   1:  PR[91,1] = PR[90,1] + -4.688;
   1:  PR[91,2] = PR[90,2] + 19.334;
   1:  PR[91,3] = PR[90,3] + 39.259;
   1:L PR[91] R[100]mm/sec CNT100;
   1:  PR[91,1] = PR[90,1] + -5.693;
   1:  PR[91,2] = PR[90,2] + 19.538;
   1:  PR[91,3] = PR[90,3] + 39.268;
   1:L PR[91] R[100]mm/sec CNT100;
   1:  PR[91,1] = PR[90,1] + -6.706;
   1:  PR[91,2] = PR[90,2] + 19.692;
   1:  PR[91,3] = PR[90,3] + 39.276;
   1:L PR[91] R[100]mm/sec CNT100;
   1:  PR[91,1] = PR[90,1] + -7.722;
   1:  PR[91,2] = PR[90,2] + 19.796;
   1:  PR[91,3] = PR[90,3] + 39.284;
   1:L PR[91] R[100]mm/sec CNT100;
   1:  PR[91,1] = PR[90,1] + -8.602;
   1:  PR[91,2] = PR[90,2] + 19.845;
   1:  PR[91,3] = PR[90,3] + 39.293;
   1:L PR[91] R[100]mm/sec CNT100;
   1:  PR[91,1] = PR[90,1] + -9.755;
   1:  PR[91,2] = PR[90,2] + 19.856;
   1:  PR[91,3] = PR[90,3] + 39.300;
   1:L PR[91] R[100]mm/sec CNT100;
   1:  PR[91,1] = PR[90,1] + -10.765;
   1:  PR[91,2] = PR[90,2] + 19.813;
   1:  PR[91,3] = PR[90,3] + 39.309;
   1:L PR[91] R[100]mm/sec CNT100;
   1:  PR[91,1] = PR[90,1] + -11.780;
   1:  PR[91,2] = PR[90,2] + 19.722;
   1:  PR[91,3] = PR[90,3] + 39.317;
   1:L PR[91] R[100]mm/sec CNT100;
   1:  PR[91,1] = PR[90,1] + -12.791;
   1:  PR[91,2] = PR[90,2] + 19.583;
   1:  PR[91,3] = PR[90,3] + 39.326;
   1:L PR[91] R[100]mm/sec CNT100;
   1:  PR[91,1] = PR[90,1] + -13.793;
   1:  PR[91,2] = PR[90,2] + 19.395;
   1:  PR[91,3] = PR[90,3] + 39.334;
   1:L PR[91] R[100]mm/sec CNT100;
   1:  PR[91,1] = PR[90,1] + -14.785;
   1:  PR[91,2] = PR[90,2] + 19.159;
   1:  PR[91,3] = PR[90,3] + 39.342;
   1:L PR[91] R[100]mm/sec CNT100;
   1:  PR[91,1] = PR[90,1] + -15.762;
   1:  PR[91,2] = PR[90,2] + 18.876;
   1:  PR[91,3] = PR[90,3] + 39.351;
   1:L PR[91] R[100]mm/sec CNT100;
   1:  PR[91,1] = PR[90,1] + -16.724;
   1:  PR[91,2] = PR[90,2] + 18.547;
   1:  PR[91,3] = PR[90,3] + 39.359;
   1:L PR[91] R[100]mm/sec CNT100;
   1:  PR[91,1] = PR[90,1] + -17.668;
   1:  PR[91,2] = PR[90,2] + 18.171;
   1:  PR[91,3] = PR[90,3] + 39.367;
   1:L PR[91] R[100]mm/sec CNT100;
   1:  PR[91,1] = PR[90,1] + -18.592;
   1:  PR[91,2] = PR[90,2] + 17.751;
   1:  PR[91,3] = PR[90,3] + 39.376;
   1:L PR[91] R[100]mm/sec CNT100;
   1:  PR[91,1] = PR[90,1] + -19.012;
   1:  PR[91,2] = PR[90,2] + 17.536;
   1:  PR[91,3] = PR[90,3] + 39.384;
   1:L PR[91] R[100]mm/sec CNT100;
   1:  PR[91,1] = PR[90,1] + -19.490;
   1:  PR[91,2] = PR[90,2] + 17.288;
   1:  PR[91,3] = PR[90,3] + 39.388;
   1:L PR[91] R[100]mm/sec CNT100;
   1:  PR[91,1] = PR[90,1] + -20.365;
   1:  PR[91,2] = PR[90,2] + 16.783;
   1:  PR[91,3] = PR[90,3] + 39.392;
   1:L PR[91] R[100]mm/sec CNT100;
   1:  PR[91,1] = PR[90,1] + -21.213;
   1:  PR[91,2] = PR[90,2] + 16.237;
   1:  PR[91,3] = PR[90,3] + 39.400;
   1:L PR[91] R[100]mm/sec CNT100;
   1:  PR[91,1] = PR[90,1] + -22.030;
   1:  PR[91,2] = PR[90,2] + 15.652;
   1:  PR[91,3] = PR[90,3] + 39.409;
   1:L PR[91] R[100]mm/sec CNT100;
   1:  PR[91,1] = PR[90,1] + -22.816;
   1:  PR[91,2] = PR[90,2] + 15.029;
   1:  PR[91,3] = PR[90,3] + 39.417;
   1:L PR[91] R[100]mm/sec CNT100;
   1:  PR[91,1] = PR[90,1] + -23.567;
   1:  PR[91,2] = PR[90,2] + 14.370;
   1:  PR[91,3] = PR[90,3] + 39.425;
   1:L PR[91] R[100]mm/sec CNT100;
   1:  PR[91,1] = PR[90,1] + -24.283;
   1:  PR[91,2] = PR[90,2] + 13.676;
   1:  PR[91,3] = PR[90,3] + 39.433;
   1:L PR[91] R[100]mm/sec CNT100;
   1:  PR[91,1] = PR[90,1] + -24.962;
   1:  PR[91,2] = PR[90,2] + 12.948;
   1:  PR[91,3] = PR[90,3] + 39.441;
   1:L PR[91] R[100]mm/sec CNT100;
   1:  PR[91,1] = PR[90,1] + -25.602;
   1:  PR[91,2] = PR[90,2] + 12.188;
   1:  PR[91,3] = PR[90,3] + 39.449;
   1:L PR[91] R[100]mm/sec CNT100;
   1:  PR[91,1] = PR[90,1] + -26.200;
   1:  PR[91,2] = PR[90,2] + 11.396;
   1:  PR[91,3] = PR[90,3] + 39.457;
   1:L PR[91] R[100]mm/sec CNT100;
   1:  PR[91,1] = PR[90,1] + -26.757;
   1:  PR[91,2] = PR[90,2] + 10.575;
   1:  PR[91,3] = PR[90,3] + 39.466;
   1:L PR[91] R[100]mm/sec CNT100;
   1:  PR[91,1] = PR[90,1] + -27.272;
   1:  PR[91,2] = PR[90,2] + 9.727;
   1:  PR[91,3] = PR[90,3] + 39.474;
   1:L PR[91] R[100]mm/sec CNT100;
   1:  PR[91,1] = PR[90,1] + -27.740;
   1:  PR[91,2] = PR[90,2] + 8.860;
   1:  PR[91,3] = PR[90,3] + 39.482;
   1:L PR[91] R[100]mm/sec CNT100;
   1:  PR[91,1] = PR[90,1] + -28.164;
   1:  PR[91,2] = PR[90,2] + 7.973;
   1:  PR[91,3] = PR[90,3] + 39.490;
   1:L PR[91] R[100]mm/sec CNT100;
   1:  PR[91,1] = PR[90,1] + -28.541;
   1:  PR[91,2] = PR[90,2] + 7.075;
   1:  PR[91,3] = PR[90,3] + 39.498;
   1:L PR[91] R[100]mm/sec CNT100;
   1:  PR[91,1] = PR[90,1] + -28.868;
   1:  PR[91,2] = PR[90,2] + 6.168;
   1:  PR[91,3] = PR[90,3] + 39.506;
   1:L PR[91] R[100]mm/sec CNT100;
   1:  PR[91,1] = PR[90,1] + -29.147;
   1:  PR[91,2] = PR[90,2] + 5.252;
   1:  PR[91,3] = PR[90,3] + 39.514;
   1:L PR[91] R[100]mm/sec CNT100;
   1:  PR[91,1] = PR[90,1] + -29.376;
   1:  PR[91,2] = PR[90,2] + 4.327;
   1:  PR[91,3] = PR[90,3] + 39.521;
   1:L PR[91] R[100]mm/sec CNT100;
   1:  PR[91,1] = PR[90,1] + -29.554;
   1:  PR[91,2] = PR[90,2] + 3.388;
   1:  PR[91,3] = PR[90,3] + 39.529;
   1:L PR[91] R[100]mm/sec CNT100;
   1:  PR[91,1] = PR[90,1] + -29.682;
   1:  PR[91,2] = PR[90,2] + 2.429;
   1:  PR[91,3] = PR[90,3] + 39.537;
   1:L PR[91] R[100]mm/sec CNT100;
   1:  PR[91,1] = PR[90,1] + -29.759;
   1:  PR[91,2] = PR[90,2] + 1.444;
   1:  PR[91,3] = PR[90,3] + 39.545;
   1:L PR[91] R[100]mm/sec CNT100;
   1:  PR[91,1] = PR[90,1] + -29.785;
   1:  PR[91,2] = PR[90,2] + 0.428;
   1:  PR[91,3] = PR[90,3] + 39.553;
   1:L PR[91] R[100]mm/sec CNT100;
   1:  PR[91,1] = PR[90,1] + -29.759;
   1:  PR[91,2] = PR[90,2] + -0.589;
   1:  PR[91,3] = PR[90,3] + 39.561;
   1:L PR[91] R[100]mm/sec CNT100;
   1:  PR[91,1] = PR[90,1] + -29.682;
   1:  PR[91,2] = PR[90,2] + -1.574;
   1:  PR[91,3] = PR[90,3] + 39.569;
   1:L PR[91] R[100]mm/sec CNT100;
   1:  PR[91,1] = PR[90,1] + -29.554;
   1:  PR[91,2] = PR[90,2] + -2.533;
   1:  PR[91,3] = PR[90,3] + 39.578;
   1:L PR[91] R[100]mm/sec CNT100;
   1:  PR[91,1] = PR[90,1] + -29.376;
   1:  PR[91,2] = PR[90,2] + -3.472;
   1:  PR[91,3] = PR[90,3] + 39.585;
   1:L PR[91] R[100]mm/sec CNT100;
   1:  PR[91,1] = PR[90,1] + -29.147;
   1:  PR[91,2] = PR[90,2] + -4.396;
   1:  PR[91,3] = PR[90,3] + 39.593;
   1:L PR[91] R[100]mm/sec CNT100;
   1:  PR[91,1] = PR[90,1] + -28.869;
   1:  PR[91,2] = PR[90,2] + -5.312;
   1:  PR[91,3] = PR[90,3] + 39.601;
   1:L PR[91] R[100]mm/sec CNT100;
   1:  PR[91,1] = PR[90,1] + -28.541;
   1:  PR[91,2] = PR[90,2] + -6.219;
   1:  PR[91,3] = PR[90,3] + 39.609;
   1:L PR[91] R[100]mm/sec CNT100;
   1:  PR[91,1] = PR[90,1] + -28.164;
   1:  PR[91,2] = PR[90,2] + -7.118;
   1:  PR[91,3] = PR[90,3] + 39.617;
   1:L PR[91] R[100]mm/sec CNT100;
   1:  PR[91,1] = PR[90,1] + -27.741;
   1:  PR[91,2] = PR[90,2] + -8.004;
   1:  PR[91,3] = PR[90,3] + 39.625;
   1:L PR[91] R[100]mm/sec CNT100;
   1:  PR[91,1] = PR[90,1] + -27.271;
   1:  PR[91,2] = PR[90,2] + -8.872;
   1:  PR[91,3] = PR[90,3] + 39.633;
   1:L PR[91] R[100]mm/sec CNT100;
   1:  PR[91,1] = PR[90,1] + -26.758;
   1:  PR[91,2] = PR[90,2] + -9.720;
   1:  PR[91,3] = PR[90,3] + 39.641;
   1:L PR[91] R[100]mm/sec CNT100;
   1:  PR[91,1] = PR[90,1] + -26.201;
   1:  PR[91,2] = PR[90,2] + -10.540;
   1:  PR[91,3] = PR[90,3] + 39.649;
   1:L PR[91] R[100]mm/sec CNT100;
   1:  PR[91,1] = PR[90,1] + -25.602;
   1:  PR[91,2] = PR[90,2] + -11.332;
   1:  PR[91,3] = PR[90,3] + 39.657;
   1:L PR[91] R[100]mm/sec CNT100;
   1:  PR[91,1] = PR[90,1] + -24.963;
   1:  PR[91,2] = PR[90,2] + -12.092;
   1:  PR[91,3] = PR[90,3] + 39.665;
   1:L PR[91] R[100]mm/sec CNT100;
   1:  PR[91,1] = PR[90,1] + -24.286;
   1:  PR[91,2] = PR[90,2] + -12.818;
   1:  PR[91,3] = PR[90,3] + 39.673;
   1:L PR[91] R[100]mm/sec CNT100;
   1:  PR[91,1] = PR[90,1] + -23.372;
   1:  PR[91,2] = PR[90,2] + -13.688;
   1:  PR[91,3] = PR[90,3] + 39.681;
   1:L PR[91] R[100]mm/sec CNT100;
   1:  PR[91,1] = PR[90,1] + -22.817;
   1:  PR[91,2] = PR[90,2] + -14.173;
   1:  PR[91,3] = PR[90,3] + 39.691;
   1:L PR[91] R[100]mm/sec CNT100;
   1:  PR[91,1] = PR[90,1] + -22.031;
   1:  PR[91,2] = PR[90,2] + -14.796;
   1:  PR[91,3] = PR[90,3] + 39.697;
   1:L PR[91] R[100]mm/sec CNT100;
   1:  PR[91,1] = PR[90,1] + -21.214;
   1:  PR[91,2] = PR[90,2] + -15.381;
   1:  PR[91,3] = PR[90,3] + 39.706;
   1:L PR[91] R[100]mm/sec CNT100;
   1:  PR[91,1] = PR[90,1] + -20.366;
   1:  PR[91,2] = PR[90,2] + -15.927;
   1:  PR[91,3] = PR[90,3] + 39.714;
   1:L PR[91] R[100]mm/sec CNT100;
   1:  PR[91,1] = PR[90,1] + -19.491;
   1:  PR[91,2] = PR[90,2] + -16.433;
   1:  PR[91,3] = PR[90,3] + 39.722;
   1:L PR[91] R[100]mm/sec CNT100;
   1:  PR[91,1] = PR[90,1] + -19.014;
   1:  PR[91,2] = PR[90,2] + -16.681;
   1:  PR[91,3] = PR[90,3] + 39.730;
   1:L PR[91] R[100]mm/sec CNT100;
   1:  PR[91,1] = PR[90,1] + -18.593;
   1:  PR[91,2] = PR[90,2] + -16.895;
   1:  PR[91,3] = PR[90,3] + 39.735;
   1:L PR[91] R[100]mm/sec CNT100;
   1:  PR[91,1] = PR[90,1] + -17.669;
   1:  PR[91,2] = PR[90,2] + -17.316;
   1:  PR[91,3] = PR[90,3] + 39.738;
   1:L PR[91] R[100]mm/sec CNT100;
   1:  PR[91,1] = PR[90,1] + -16.726;
   1:  PR[91,2] = PR[90,2] + -17.691;
   1:  PR[91,3] = PR[90,3] + 39.747;
   1:L PR[91] R[100]mm/sec CNT100;
   1:  PR[91,1] = PR[90,1] + -15.764;
   1:  PR[91,2] = PR[90,2] + -18.021;
   1:  PR[91,3] = PR[90,3] + 39.755;
   1:L PR[91] R[100]mm/sec CNT100;
   1:  PR[91,1] = PR[90,1] + -14.786;
   1:  PR[91,2] = PR[90,2] + -18.304;
   1:  PR[91,3] = PR[90,3] + 39.763;
   1:L PR[91] R[100]mm/sec CNT100;
   1:  PR[91,1] = PR[90,1] + -13.795;
   1:  PR[91,2] = PR[90,2] + -18.539;
   1:  PR[91,3] = PR[90,3] + 39.772;
   1:L PR[91] R[100]mm/sec CNT100;
   1:  PR[91,1] = PR[90,1] + -12.792;
   1:  PR[91,2] = PR[90,2] + -18.727;
   1:  PR[91,3] = PR[90,3] + 39.780;
   1:L PR[91] R[100]mm/sec CNT100;
   1:  PR[91,1] = PR[90,1] + -11.781;
   1:  PR[91,2] = PR[90,2] + -18.867;
   1:  PR[91,3] = PR[90,3] + 39.788;
   1:L PR[91] R[100]mm/sec CNT100;
   1:  PR[91,1] = PR[90,1] + -10.754;
   1:  PR[91,2] = PR[90,2] + -18.958;
   1:  PR[91,3] = PR[90,3] + 39.797;
   1:L PR[91] R[100]mm/sec CNT100;
   1:  PR[91,1] = PR[90,1] + -9.755;
   1:  PR[91,2] = PR[90,2] + -19.001;
   1:  PR[91,3] = PR[90,3] + 39.805;
   1:L PR[91] R[100]mm/sec CNT100;
   1:  PR[91,1] = PR[90,1] + -8.740;
   1:  PR[91,2] = PR[90,2] + -18.995;
   1:  PR[91,3] = PR[90,3] + 39.813;
   1:L PR[91] R[100]mm/sec CNT100;
   1:  PR[91,1] = PR[90,1] + -7.723;
   1:  PR[91,2] = PR[90,2] + -18.941;
   1:  PR[91,3] = PR[90,3] + 39.821;
   1:L PR[91] R[100]mm/sec CNT100;
   1:  PR[91,1] = PR[90,1] + -6.707;
   1:  PR[91,2] = PR[90,2] + -18.837;
   1:  PR[91,3] = PR[90,3] + 39.830;
   1:L PR[91] R[100]mm/sec CNT100;
   1:  PR[91,1] = PR[90,1] + -5.695;
   1:  PR[91,2] = PR[90,2] + -18.683;
   1:  PR[91,3] = PR[90,3] + 39.838;
   1:L PR[91] R[100]mm/sec CNT100;
   1:  PR[91,1] = PR[90,1] + -4.689;
   1:  PR[91,2] = PR[90,2] + -18.479;
   1:  PR[91,3] = PR[90,3] + 39.846;
   1:L PR[91] R[100]mm/sec CNT100;
   1:  PR[91,1] = PR[90,1] + -3.692;
   1:  PR[91,2] = PR[90,2] + -18.226;
   1:  PR[91,3] = PR[90,3] + 39.855;
   1:L PR[91] R[100]mm/sec CNT100;
   1:  PR[91,1] = PR[90,1] + -2.707;
   1:  PR[91,2] = PR[90,2] + -17.922;
   1:  PR[91,3] = PR[90,3] + 39.863;
   1:L PR[91] R[100]mm/sec CNT100;
   1:  PR[91,1] = PR[90,1] + -1.736;
   1:  PR[91,2] = PR[90,2] + -17.569;
   1:  PR[91,3] = PR[90,3] + 39.872;
   1:L PR[91] R[100]mm/sec CNT100;
   1:  PR[91,1] = PR[90,1] + -1.258;
   1:  PR[91,2] = PR[90,2] + -17.370;
   1:  PR[91,3] = PR[90,3] + 39.880;
   1:L PR[91] R[100]mm/sec CNT100;
   1:  PR[91,1] = PR[90,1] + -0.818;
   1:  PR[91,2] = PR[90,2] + -17.224;
   1:  PR[91,3] = PR[90,3] + 39.884;
   1:L PR[91] R[100]mm/sec CNT100;
   1:  PR[91,1] = PR[90,1] + -0.333;
   1:  PR[91,2] = PR[90,2] + -17.149;
   1:  PR[91,3] = PR[90,3] + 39.888;
   1:L PR[91] R[100]mm/sec CNT100;
   1:  PR[91,1] = PR[90,1] + 0.158;
   1:  PR[91,2] = PR[90,2] + -17.154;
   1:  PR[91,3] = PR[90,3] + 39.892;
   1:L PR[91] R[100]mm/sec CNT100;
   1:  PR[91,1] = PR[90,1] + 0.648;
   1:  PR[91,2] = PR[90,2] + -17.241;
   1:  PR[91,3] = PR[90,3] + 39.896;
   1:L PR[91] R[100]mm/sec CNT100;
   1:  PR[91] = PR[90];
   1:  PR[91,1] = PR[90,1] + 2.126;
   1:  PR[91,2] = PR[90,2] + -18.183;
   1:  PR[91,3] = PR[90,3] + 41.230;
   1:L PR[91] R[100]mm/sec CNT100;
   1:  PR[91,1] = PR[90,1] + 3.017;
   1:  PR[91,2] = PR[90,2] + -18.451;
   1:  PR[91,3] = PR[90,3] + 39.912;
   1:L PR[91] R[100]mm/sec CNT100;
   1:  PR[91,1] = PR[90,1] + 4.031;
   1:  PR[91,2] = PR[90,2] + -18.704;
   1:  PR[91,3] = PR[90,3] + 39.920;
   1:L PR[91] R[100]mm/sec CNT100;
   1:  PR[91,1] = PR[90,1] + 5.334;
   1:  PR[91,2] = PR[90,2] + -18.949;
   1:  PR[91,3] = PR[90,3] + 39.929;
   1:L PR[91] R[100]mm/sec CNT100;
   1:  PR[91,1] = PR[90,1] + 6.089;
   1:  PR[91,2] = PR[90,2] + -19.055;
   1:  PR[91,3] = PR[90,3] + 39.939;
   1:L PR[91] R[100]mm/sec CNT100;
   1:  PR[91,1] = PR[90,1] + 7.125;
   1:  PR[91,2] = PR[90,2] + -19.154;
   1:  PR[91,3] = PR[90,3] + 39.946;
   1:L PR[91] R[100]mm/sec CNT100;
   1:  PR[91,1] = PR[90,1] + 8.161;
   1:  PR[91,2] = PR[90,2] + -19.201;
   1:  PR[91,3] = PR[90,3] + 39.954;
   1:L PR[91] R[100]mm/sec CNT100;
   1:  PR[91,1] = PR[90,1] + 9.195;
   1:  PR[91,2] = PR[90,2] + -19.198;
   1:  PR[91,3] = PR[90,3] + 39.963;
   1:L PR[91] R[100]mm/sec CNT100;
   1:  PR[91,1] = PR[90,1] + 10.227;
   1:  PR[91,2] = PR[90,2] + -19.145;
   1:  PR[91,3] = PR[90,3] + 39.971;
   1:L PR[91] R[100]mm/sec CNT100;
   1:  PR[91,1] = PR[90,1] + 10.777;
   1:  PR[91,2] = PR[90,2] + -19.095;
   1:  PR[91,3] = PR[90,3] + 39.980;
   1:L PR[91] R[100]mm/sec CNT100;
   1:  PR[91,1] = PR[90,1] + 11.243;
   1:  PR[91,2] = PR[90,2] + -19.043;
   1:  PR[91,3] = PR[90,3] + 39.984;
   1:L PR[91] R[100]mm/sec CNT100;
   1:  PR[91,1] = PR[90,1] + 12.258;
   1:  PR[91,2] = PR[90,2] + -18.891;
   1:  PR[91,3] = PR[90,3] + 39.988;
   1:L PR[91] R[100]mm/sec CNT100;
   1:  PR[91,1] = PR[90,1] + 13.258;
   1:  PR[91,2] = PR[90,2] + -18.692;
   1:  PR[91,3] = PR[90,3] + 39.997;
   1:L PR[91] R[100]mm/sec CNT100;
   1:  PR[91,1] = PR[90,1] + 14.244;
   1:  PR[91,2] = PR[90,2] + -18.447;
   1:  PR[91,3] = PR[90,3] + 40.005;
   1:L PR[91] R[100]mm/sec CNT100;
   1:  PR[91,1] = PR[90,1] + 15.213;
   1:  PR[91,2] = PR[90,2] + -18.155;
   1:  PR[91,3] = PR[90,3] + 40.013;
   1:L PR[91] R[100]mm/sec CNT100;
   1:  PR[91,1] = PR[90,1] + 16.164;
   1:  PR[91,2] = PR[90,2] + -17.820;
   1:  PR[91,3] = PR[90,3] + 40.022;
   1:L PR[91] R[100]mm/sec CNT100;
   1:  PR[91,1] = PR[90,1] + 16.987;
   1:  PR[91,2] = PR[90,2] + -17.488;
   1:  PR[91,3] = PR[90,3] + 40.030;
   1:L PR[91] R[100]mm/sec CNT100;
   1:  PR[91,1] = PR[90,1] + 17.948;
   1:  PR[91,2] = PR[90,2] + -17.047;
   1:  PR[91,3] = PR[90,3] + 40.037;
   1:L PR[91] R[100]mm/sec CNT100;
   1:  PR[91,1] = PR[90,1] + 18.881;
   1:  PR[91,2] = PR[90,2] + -16.562;
   1:  PR[91,3] = PR[90,3] + 40.046;
   1:L PR[91] R[100]mm/sec CNT100;
   1:  PR[91,1] = PR[90,1] + 19.757;
   1:  PR[91,2] = PR[90,2] + -16.051;
   1:  PR[91,3] = PR[90,3] + 40.054;
   1:L PR[91] R[100]mm/sec CNT100;
   1:  PR[91,1] = PR[90,1] + 20.606;
   1:  PR[91,2] = PR[90,2] + -15.500;
   1:  PR[91,3] = PR[90,3] + 40.063;
   1:L PR[91] R[100]mm/sec CNT100;
   1:  PR[91,1] = PR[90,1] + 21.424;
   1:  PR[91,2] = PR[90,2] + -14.910;
   1:  PR[91,3] = PR[90,3] + 40.071;
   1:L PR[91] R[100]mm/sec CNT100;
   1:  PR[91,1] = PR[90,1] + 22.211;
   1:  PR[91,2] = PR[90,2] + -14.281;
   1:  PR[91,3] = PR[90,3] + 40.079;
   1:L PR[91] R[100]mm/sec CNT100;
   1:  PR[91,1] = PR[90,1] + 22.964;
   1:  PR[91,2] = PR[90,2] + -13.615;
   1:  PR[91,3] = PR[90,3] + 40.088;
   1:L PR[91] R[100]mm/sec CNT100;
   1:  PR[91,1] = PR[90,1] + 23.681;
   1:  PR[91,2] = PR[90,2] + -12.913;
   1:  PR[91,3] = PR[90,3] + 40.096;
   1:L PR[91] R[100]mm/sec CNT100;
   1:  PR[91,1] = PR[90,1] + 24.360;
   1:  PR[91,2] = PR[90,2] + -12.177;
   1:  PR[91,3] = PR[90,3] + 40.104;
   1:L PR[91] R[100]mm/sec CNT100;
   1:  PR[91,1] = PR[90,1] + 25.001;
   1:  PR[91,2] = PR[90,2] + -11.408;
   1:  PR[91,3] = PR[90,3] + 40.112;
   1:L PR[91] R[100]mm/sec CNT100;
   1:  PR[91,1] = PR[90,1] + 25.600;
   1:  PR[91,2] = PR[90,2] + -10.608;
   1:  PR[91,3] = PR[90,3] + 40.121;
   1:L PR[91] R[100]mm/sec CNT100;
   1:  PR[91,1] = PR[90,1] + 26.158;
   1:  PR[91,2] = PR[90,2] + -9.780;
   1:  PR[91,3] = PR[90,3] + 40.129;
   1:L PR[91] R[100]mm/sec CNT100;
   1:  PR[91,1] = PR[90,1] + 26.393;
   1:  PR[91,2] = PR[90,2] + -9.394;
   1:  PR[91,3] = PR[90,3] + 40.137;
   1:L PR[91] R[100]mm/sec CNT100;
   1:  PR[91,1] = PR[90,1] + 26.672;
   1:  PR[91,2] = PR[90,2] + -8.930;
   1:  PR[91,3] = PR[90,3] + 40.141;
   1:L PR[91] R[100]mm/sec CNT100;
   1:  PR[91,1] = PR[90,1] + 27.142;
   1:  PR[91,2] = PR[90,2] + -8.057;
   1:  PR[91,3] = PR[90,3] + 40.145;
   1:L PR[91] R[100]mm/sec CNT100;
   1:  PR[91,1] = PR[90,1] + 27.565;
   1:  PR[91,2] = PR[90,2] + -7.169;
   1:  PR[91,3] = PR[90,3] + 40.153;
   1:L PR[91] R[100]mm/sec CNT100;
   1:  PR[91,1] = PR[90,1] + 27.941;
   1:  PR[91,2] = PR[90,2] + -6.269;
   1:  PR[91,3] = PR[90,3] + 40.161;
   1:L PR[91] R[100]mm/sec CNT100;
   1:  PR[91,1] = PR[90,1] + 28.268;
   1:  PR[91,2] = PR[90,2] + -5.359;
   1:  PR[91,3] = PR[90,3] + 40.169;
   1:L PR[91] R[100]mm/sec CNT100;
   1:  PR[91,1] = PR[90,1] + 28.546;
   1:  PR[91,2] = PR[90,2] + -4.438;
   1:  PR[91,3] = PR[90,3] + 40.177;
   1:L PR[91] R[100]mm/sec CNT100;
   1:  PR[91,1] = PR[90,1] + 28.774;
   1:  PR[91,2] = PR[90,2] + -3.505;
   1:  PR[91,3] = PR[90,3] + 40.185;
   1:L PR[91] R[100]mm/sec CNT100;
   1:  PR[91,1] = PR[90,1] + 28.952;
   1:  PR[91,2] = PR[90,2] + -2.556;
   1:  PR[91,3] = PR[90,3] + 40.193;
   1:L PR[91] R[100]mm/sec CNT100;
   1:  PR[91,1] = PR[90,1] + 29.080;
   1:  PR[91,2] = PR[90,2] + -1.586;
   1:  PR[91,3] = PR[90,3] + 40.201;
   1:L PR[91] R[100]mm/sec CNT100;
   1:  PR[91,1] = PR[90,1] + 29.157;
   1:  PR[91,2] = PR[90,2] + -0.593;
   1:  PR[91,3] = PR[90,3] + 40.209;
   1:L PR[91] R[100]mm/sec CNT100;
   1:  PR[91,1] = PR[90,1] + 29.181;
   1:  PR[91,2] = PR[90,2] + 0.428;
   1:  PR[91,3] = PR[90,3] + 40.217;
   1:L PR[91] R[100]mm/sec CNT100;
   1:  PR[91,1] = PR[90,1] + 29.157;
   1:  PR[91,2] = PR[90,2] + 1.448;
   1:  PR[91,3] = PR[90,3] + 40.226;
   1:L PR[91] R[100]mm/sec CNT100;
   1:  PR[91,1] = PR[90,1] + 29.080;
   1:  PR[91,2] = PR[90,2] + 2.441;
   1:  PR[91,3] = PR[90,3] + 40.234;
   1:L PR[91] R[100]mm/sec CNT100;
   1:  PR[91,1] = PR[90,1] + 28.952;
   1:  PR[91,2] = PR[90,2] + 3.411;
   1:  PR[91,3] = PR[90,3] + 40.242;
   1:L PR[91] R[100]mm/sec CNT100;
   1:  PR[91,1] = PR[90,1] + 28.774;
   1:  PR[91,2] = PR[90,2] + 4.360;
   1:  PR[91,3] = PR[90,3] + 40.250;
   1:L PR[91] R[100]mm/sec CNT100;
   1:  PR[91,1] = PR[90,1] + 28.546;
   1:  PR[91,2] = PR[90,2] + 5.294;
   1:  PR[91,3] = PR[90,3] + 40.258;
   1:L PR[91] R[100]mm/sec CNT100;
   1:  PR[91,1] = PR[90,1] + 28.268;
   1:  PR[91,2] = PR[90,2] + 6.215;
   1:  PR[91,3] = PR[90,3] + 40.266;
   1:L PR[91] R[100]mm/sec CNT100;
   1:  PR[91,1] = PR[90,1] + 27.941;
   1:  PR[91,2] = PR[90,2] + 7.125;
   1:  PR[91,3] = PR[90,3] + 40.274;
   1:L PR[91] R[100]mm/sec CNT100;
   1:  PR[91,1] = PR[90,1] + 27.771;
   1:  PR[91,2] = PR[90,2] + 7.533;
   1:  PR[91,3] = PR[90,3] + 40.282;
   1:L PR[91] R[100]mm/sec CNT100;
   1:  PR[91,1] = PR[90,1] + 27.565;
   1:  PR[91,2] = PR[90,2] + 8.024;
   1:  PR[91,3] = PR[90,3] + 40.285;
   1:L PR[91] R[100]mm/sec CNT100;
   1:  PR[91,1] = PR[90,1] + 27.141;
   1:  PR[91,2] = PR[90,2] + 8.913;
   1:  PR[91,3] = PR[90,3] + 40.290;
   1:L PR[91] R[100]mm/sec CNT100;
   1:  PR[91,1] = PR[90,1] + 26.672;
   1:  PR[91,2] = PR[90,2] + 9.785;
   1:  PR[91,3] = PR[90,3] + 40.298;
   1:L PR[91] R[100]mm/sec CNT100;
   1:  PR[91,1] = PR[90,1] + 26.158;
   1:  PR[91,2] = PR[90,2] + 10.636;
   1:  PR[91,3] = PR[90,3] + 40.306;
   1:L PR[91] R[100]mm/sec CNT100;
   1:  PR[91,1] = PR[90,1] + 25.600;
   1:  PR[91,2] = PR[90,2] + 11.464;
   1:  PR[91,3] = PR[90,3] + 40.314;
   1:L PR[91] R[100]mm/sec CNT100;
   1:  PR[91,1] = PR[90,1] + 25.230;
   1:  PR[91,2] = PR[90,2] + 11.960;
   1:  PR[91,3] = PR[90,3] + 40.322;
   1:L PR[91] R[100]mm/sec CNT100;
   1:  PR[91,1] = PR[90,1] + 25.001;
   1:  PR[91,2] = PR[90,2] + 12.263;
   1:  PR[91,3] = PR[90,3] + 40.328;
   1:L PR[91] R[100]mm/sec CNT100;
   1:  PR[91,1] = PR[90,1] + 24.360;
   1:  PR[91,2] = PR[90,2] + 13.032;
   1:  PR[91,3] = PR[90,3] + 40.331;
   1:L PR[91] R[100]mm/sec CNT100;
   1:  PR[91,1] = PR[90,1] + 23.680;
   1:  PR[91,2] = PR[90,2] + 13.768;
   1:  PR[91,3] = PR[90,3] + 40.339;
   1:L PR[91] R[100]mm/sec CNT100;
   1:  PR[91,1] = PR[90,1] + 22.963;
   1:  PR[91,2] = PR[90,2] + 14.471;
   1:  PR[91,3] = PR[90,3] + 40.347;
   1:L PR[91] R[100]mm/sec CNT100;
   1:  PR[91,1] = PR[90,1] + 22.210;
   1:  PR[91,2] = PR[90,2] + 15.136;
   1:  PR[91,3] = PR[90,3] + 40.355;
   1:L PR[91] R[100]mm/sec CNT100;
   1:  PR[91,1] = PR[90,1] + 21.549;
   1:  PR[91,2] = PR[90,2] + 15.666;
   1:  PR[91,3] = PR[90,3] + 40.364;
   1:L PR[91] R[100]mm/sec CNT100;
   1:  PR[91,1] = PR[90,1] + 20.603;
   1:  PR[91,2] = PR[90,2] + 16.357;
   1:  PR[91,3] = PR[90,3] + 40.371;
   1:L PR[91] R[100]mm/sec CNT100;
   1:  PR[91,1] = PR[90,1] + 19.756;
   1:  PR[91,2] = PR[90,2] + 16.907;
   1:  PR[91,3] = PR[90,3] + 40.380;
   1:L PR[91] R[100]mm/sec CNT100;
   1:  PR[91,1] = PR[90,1] + 18.879;
   1:  PR[91,2] = PR[90,2] + 17.418;
   1:  PR[91,3] = PR[90,3] + 40.388;
   1:L PR[91] R[100]mm/sec CNT100;
   1:  PR[91,1] = PR[90,1] + 17.947;
   1:  PR[91,2] = PR[90,2] + 17.903;
   1:  PR[91,3] = PR[90,3] + 40.397;
   1:L PR[91] R[100]mm/sec CNT100;
   1:  PR[91,1] = PR[90,1] + 16.986;
   1:  PR[91,2] = PR[90,2] + 18.343;
   1:  PR[91,3] = PR[90,3] + 40.405;
   1:L PR[91] R[100]mm/sec CNT100;
   1:  PR[91,1] = PR[90,1] + 16.163;
   1:  PR[91,2] = PR[90,2] + 18.675;
   1:  PR[91,3] = PR[90,3] + 40.414;
   1:L PR[91] R[100]mm/sec CNT100;
   1:  PR[91,1] = PR[90,1] + 15.212;
   1:  PR[91,2] = PR[90,2] + 19.011;
   1:  PR[91,3] = PR[90,3] + 40.421;
   1:L PR[91] R[100]mm/sec CNT100;
   1:  PR[91,1] = PR[90,1] + 14.243;
   1:  PR[91,2] = PR[90,2] + 19.302;
   1:  PR[91,3] = PR[90,3] + 40.430;
   1:L PR[91] R[100]mm/sec CNT100;
   1:  PR[91,1] = PR[90,1] + 13.257;
   1:  PR[91,2] = PR[90,2] + 19.548;
   1:  PR[91,3] = PR[90,3] + 40.438;
   1:L PR[91] R[100]mm/sec CNT100;
   1:  PR[91,1] = PR[90,1] + 12.254;
   1:  PR[91,2] = PR[90,2] + 19.747;
   1:  PR[91,3] = PR[90,3] + 40.446;
   1:L PR[91] R[100]mm/sec CNT100;
   1:  PR[91,1] = PR[90,1] + 11.852;
   1:  PR[91,2] = PR[90,2] + 19.812;
   1:  PR[91,3] = PR[90,3] + 40.455;
   1:L PR[91] R[100]mm/sec CNT100;
   1:  PR[91,1] = PR[90,1] + 11.247;
   1:  PR[91,2] = PR[90,2] + 19.898;
   1:  PR[91,3] = PR[90,3] + 40.458;
   1:L PR[91] R[100]mm/sec CNT100;
   1:  PR[91,1] = PR[90,1] + 10.223;
   1:  PR[91,2] = PR[90,2] + 20.000;
   1:  PR[91,3] = PR[90,3] + 40.463;
   1:L PR[91] R[100]mm/sec CNT100;
   1:  PR[91,1] = PR[90,1] + 9.192;
   1:  PR[91,2] = PR[90,2] + 20.053;
   1:  PR[91,3] = PR[90,3] + 40.472;
   1:L PR[91] R[100]mm/sec CNT100;
   1:  PR[91,1] = PR[90,1] + 8.600;
   1:  PR[91,2] = PR[90,2] + 20.060;
   1:  PR[91,3] = PR[90,3] + 40.480;
   1:L PR[91] R[100]mm/sec CNT100;
   1:  PR[91,1] = PR[90,1] + 8.163;
   1:  PR[91,2] = PR[90,2] + 20.057;
   1:  PR[91,3] = PR[90,3] + 40.485;
   1:L PR[91] R[100]mm/sec CNT100;
   1:  PR[91,1] = PR[90,1] + 7.124;
   1:  PR[91,2] = PR[90,2] + 20.009;
   1:  PR[91,3] = PR[90,3] + 40.488;
   1:L PR[91] R[100]mm/sec CNT100;
   1:  PR[91,1] = PR[90,1] + 6.089;
   1:  PR[91,2] = PR[90,2] + 19.911;
   1:  PR[91,3] = PR[90,3] + 40.497;
   1:L PR[91] R[100]mm/sec CNT100;
   1:  PR[91,1] = PR[90,1] + 5.058;
   1:  PR[91,2] = PR[90,2] + 19.761;
   1:  PR[91,3] = PR[90,3] + 40.506;
   1:L PR[91] R[100]mm/sec CNT100;
   1:  PR[91,1] = PR[90,1] + 4.033;
   1:  PR[91,2] = PR[90,2] + 19.559;
   1:  PR[91,3] = PR[90,3] + 40.514;
   1:L PR[91] R[100]mm/sec CNT100;
   1:  PR[91,1] = PR[90,1] + 3.017;
   1:  PR[91,2] = PR[90,2] + 19.306;
   1:  PR[91,3] = PR[90,3] + 40.523;
   1:L PR[91] R[100]mm/sec CNT100;
   1:  PR[91,1] = PR[90,1] + 2.013;
   1:  PR[91,2] = PR[90,2] + 19.003;
   1:  PR[91,3] = PR[90,3] + 40.531;
   1:L PR[91] R[100]mm/sec CNT100;
   1:  PR[91,1] = PR[90,1] + 0.710;
   1:  PR[91,2] = PR[90,2] + 18.536;
   1:  PR[91,3] = PR[90,3] + 40.540;
   1:L PR[91] R[100]mm/sec CNT100;
   1:  PR[91,1] = PR[90,1] + 0.230;
   1:  PR[91,2] = PR[90,2] + 18.441;
   1:  PR[91,3] = PR[90,3] + 40.551;
   1:L PR[91] R[100]mm/sec CNT100;
   1:  PR[91,1] = PR[90,1] + -0.255;
   1:  PR[91,2] = PR[90,2] + 18.422;
   1:  PR[91,3] = PR[90,3] + 40.555;
   1:L PR[91] R[100]mm/sec CNT100;
   1:  PR[91,1] = PR[90,1] + -0.742;
   1:  PR[91,2] = PR[90,2] + 18.485;
   1:  PR[91,3] = PR[90,3] + 40.559;
   1:L PR[91] R[100]mm/sec CNT100;
   1:  PR[91,1] = PR[90,1] + -1.178;
   1:  PR[91,2] = PR[90,2] + 18.616;
   1:  PR[91,3] = PR[90,3] + 40.563;
   1:L PR[91] R[100]mm/sec CNT100;
   1:  PR[91,1] = PR[90,1] + -2.363;
   1:  PR[91,2] = PR[90,2] + 19.039;
   1:  PR[91,3] = PR[90,3] + 40.567;
   1:L PR[91] R[100]mm/sec CNT100;
   1:  PR[91,1] = PR[90,1] + -3.255;
   1:  PR[91,2] = PR[90,2] + 19.307;
   1:  PR[91,3] = PR[90,3] + 40.577;
   1:L PR[91] R[100]mm/sec CNT100;
   1:  PR[91,1] = PR[90,1] + -4.269;
   1:  PR[91,2] = PR[90,2] + 19.559;
   1:  PR[91,3] = PR[90,3] + 40.585;
   1:L PR[91] R[100]mm/sec CNT100;
   1:  PR[91,1] = PR[90,1] + -5.571;
   1:  PR[91,2] = PR[90,2] + 19.804;
   1:  PR[91,3] = PR[90,3] + 40.594;
   1:L PR[91] R[100]mm/sec CNT100;
   1:  PR[91,1] = PR[90,1] + -6.327;
   1:  PR[91,2] = PR[90,2] + 19.910;
   1:  PR[91,3] = PR[90,3] + 40.604;
   1:L PR[91] R[100]mm/sec CNT100;
   1:  PR[91,1] = PR[90,1] + -7.363;
   1:  PR[91,2] = PR[90,2] + 20.009;
   1:  PR[91,3] = PR[90,3] + 40.611;
   1:L PR[91] R[100]mm/sec CNT100;
   1:  PR[91,1] = PR[90,1] + -8.399;
   1:  PR[91,2] = PR[90,2] + 20.056;
   1:  PR[91,3] = PR[90,3] + 40.619;
   1:L PR[91] R[100]mm/sec CNT100;
   1:  PR[91,1] = PR[90,1] + -9.433;
   1:  PR[91,2] = PR[90,2] + 20.053;
   1:  PR[91,3] = PR[90,3] + 40.628;
   1:L PR[91] R[100]mm/sec CNT100;
   1:  PR[91,1] = PR[90,1] + -10.465;
   1:  PR[91,2] = PR[90,2] + 20.000;
   1:  PR[91,3] = PR[90,3] + 40.636;
   1:L PR[91] R[100]mm/sec CNT100;
   1:  PR[91,1] = PR[90,1] + -11.016;
   1:  PR[91,2] = PR[90,2] + 19.949;
   1:  PR[91,3] = PR[90,3] + 40.645;
   1:L PR[91] R[100]mm/sec CNT100;
   1:  PR[91,1] = PR[90,1] + -11.481;
   1:  PR[91,2] = PR[90,2] + 19.898;
   1:  PR[91,3] = PR[90,3] + 40.649;
   1:L PR[91] R[100]mm/sec CNT100;
   1:  PR[91,1] = PR[90,1] + -12.496;
   1:  PR[91,2] = PR[90,2] + 19.746;
   1:  PR[91,3] = PR[90,3] + 40.653;
   1:L PR[91] R[100]mm/sec CNT100;
   1:  PR[91,1] = PR[90,1] + -13.497;
   1:  PR[91,2] = PR[90,2] + 19.548;
   1:  PR[91,3] = PR[90,3] + 40.662;
   1:L PR[91] R[100]mm/sec CNT100;
   1:  PR[91,1] = PR[90,1] + -14.482;
   1:  PR[91,2] = PR[90,2] + 19.303;
   1:  PR[91,3] = PR[90,3] + 40.670;
   1:L PR[91] R[100]mm/sec CNT100;
   1:  PR[91,1] = PR[90,1] + -15.453;
   1:  PR[91,2] = PR[90,2] + 19.011;
   1:  PR[91,3] = PR[90,3] + 40.678;
   1:L PR[91] R[100]mm/sec CNT100;
   1:  PR[91,1] = PR[90,1] + -16.239;
   1:  PR[91,2] = PR[90,2] + 18.738;
   1:  PR[91,3] = PR[90,3] + 40.687;
   1:L PR[91] R[100]mm/sec CNT100;
   1:  PR[91,1] = PR[90,1] + -17.226;
   1:  PR[91,2] = PR[90,2] + 18.343;
   1:  PR[91,3] = PR[90,3] + 40.693;
   1:L PR[91] R[100]mm/sec CNT100;
   1:  PR[91,1] = PR[90,1] + -18.186;
   1:  PR[91,2] = PR[90,2] + 17.903;
   1:  PR[91,3] = PR[90,3] + 40.702;
   1:L PR[91] R[100]mm/sec CNT100;
   1:  PR[91,1] = PR[90,1] + -19.119;
   1:  PR[91,2] = PR[90,2] + 17.416;
   1:  PR[91,3] = PR[90,3] + 40.711;
   1:L PR[91] R[100]mm/sec CNT100;
   1:  PR[91,1] = PR[90,1] + -19.995;
   1:  PR[91,2] = PR[90,2] + 16.905;
   1:  PR[91,3] = PR[90,3] + 40.719;
   1:L PR[91] R[100]mm/sec CNT100;
   1:  PR[91,1] = PR[90,1] + -20.844;
   1:  PR[91,2] = PR[90,2] + 16.353;
   1:  PR[91,3] = PR[90,3] + 40.728;
   1:L PR[91] R[100]mm/sec CNT100;
   1:  PR[91,1] = PR[90,1] + -21.663;
   1:  PR[91,2] = PR[90,2] + 15.762;
   1:  PR[91,3] = PR[90,3] + 40.736;
   1:L PR[91] R[100]mm/sec CNT100;
   1:  PR[91,1] = PR[90,1] + -22.450;
   1:  PR[91,2] = PR[90,2] + 15.133;
   1:  PR[91,3] = PR[90,3] + 40.744;
   1:L PR[91] R[100]mm/sec CNT100;
   1:  PR[91,1] = PR[90,1] + -23.203;
   1:  PR[91,2] = PR[90,2] + 14.468;
   1:  PR[91,3] = PR[90,3] + 40.753;
   1:L PR[91] R[100]mm/sec CNT100;
   1:  PR[91,1] = PR[90,1] + -23.920;
   1:  PR[91,2] = PR[90,2] + 13.768;
   1:  PR[91,3] = PR[90,3] + 40.761;
   1:L PR[91] R[100]mm/sec CNT100;
   1:  PR[91,1] = PR[90,1] + -24.599;
   1:  PR[91,2] = PR[90,2] + 13.034;
   1:  PR[91,3] = PR[90,3] + 40.769;
   1:L PR[91] R[100]mm/sec CNT100;
   1:  PR[91,1] = PR[90,1] + -25.240;
   1:  PR[91,2] = PR[90,2] + 12.266;
   1:  PR[91,3] = PR[90,3] + 40.777;
   1:L PR[91] R[100]mm/sec CNT100;
   1:  PR[91,1] = PR[90,1] + -25.469;
   1:  PR[91,2] = PR[90,2] + 11.965;
   1:  PR[91,3] = PR[90,3] + 40.786;
   1:L PR[91] R[100]mm/sec CNT100;
   1:  PR[91,1] = PR[90,1] + -25.839;
   1:  PR[91,2] = PR[90,2] + 11.470;
   1:  PR[91,3] = PR[90,3] + 40.789;
   1:L PR[91] R[100]mm/sec CNT100;
   1:  PR[91,1] = PR[90,1] + -26.397;
   1:  PR[91,2] = PR[90,2] + 10.643;
   1:  PR[91,3] = PR[90,3] + 40.794;
   1:L PR[91] R[100]mm/sec CNT100;
   1:  PR[91,1] = PR[90,1] + -26.911;
   1:  PR[91,2] = PR[90,2] + 9.790;
   1:  PR[91,3] = PR[90,3] + 40.802;
   1:L PR[91] R[100]mm/sec CNT100;
   1:  PR[91,1] = PR[90,1] + -27.380;
   1:  PR[91,2] = PR[90,2] + 8.915;
   1:  PR[91,3] = PR[90,3] + 40.810;
   1:L PR[91] R[100]mm/sec CNT100;
   1:  PR[91,1] = PR[90,1] + -27.803;
   1:  PR[91,2] = PR[90,2] + 8.023;
   1:  PR[91,3] = PR[90,3] + 40.818;
   1:L PR[91] R[100]mm/sec CNT100;
   1:  PR[91,1] = PR[90,1] + -28.179;
   1:  PR[91,2] = PR[90,2] + 7.117;
   1:  PR[91,3] = PR[90,3] + 40.826;
   1:L PR[91] R[100]mm/sec CNT100;
   1:  PR[91,1] = PR[90,1] + -28.507;
   1:  PR[91,2] = PR[90,2] + 6.203;
   1:  PR[91,3] = PR[90,3] + 40.834;
   1:L PR[91] R[100]mm/sec CNT100;
   1:  PR[91,1] = PR[90,1] + -28.785;
   1:  PR[91,2] = PR[90,2] + 5.280;
   1:  PR[91,3] = PR[90,3] + 40.842;
   1:L PR[91] R[100]mm/sec CNT100;
   1:  PR[91,1] = PR[90,1] + -29.013;
   1:  PR[91,2] = PR[90,2] + 4.348;
   1:  PR[91,3] = PR[90,3] + 40.850;
   1:L PR[91] R[100]mm/sec CNT100;
   1:  PR[91,1] = PR[90,1] + -29.191;
   1:  PR[91,2] = PR[90,2] + 3.402;
   1:  PR[91,3] = PR[90,3] + 40.858;
   1:L PR[91] R[100]mm/sec CNT100;
   1:  PR[91,1] = PR[90,1] + -29.319;
   1:  PR[91,2] = PR[90,2] + 2.436;
   1:  PR[91,3] = PR[90,3] + 40.866;
   1:L PR[91] R[100]mm/sec CNT100;
   1:  PR[91,1] = PR[90,1] + -29.396;
   1:  PR[91,2] = PR[90,2] + 1.447;
   1:  PR[91,3] = PR[90,3] + 40.874;
   1:L PR[91] R[100]mm/sec CNT100;
   1:  PR[91,1] = PR[90,1] + -29.420;
   1:  PR[91,2] = PR[90,2] + 0.428;
   1:  PR[91,3] = PR[90,3] + 40.882;
   1:L PR[91] R[100]mm/sec CNT100;
   1:  PR[91,1] = PR[90,1] + -29.396;
   1:  PR[91,2] = PR[90,2] + -0.592;
   1:  PR[91,3] = PR[90,3] + 40.891;
   1:L PR[91] R[100]mm/sec CNT100;
   1:  PR[91,1] = PR[90,1] + -29.319;
   1:  PR[91,2] = PR[90,2] + -1.581;
   1:  PR[91,3] = PR[90,3] + 40.899;
   1:L PR[91] R[100]mm/sec CNT100;
   1:  PR[91,1] = PR[90,1] + -29.191;
   1:  PR[91,2] = PR[90,2] + -2.546;
   1:  PR[91,3] = PR[90,3] + 40.907;
   1:L PR[91] R[100]mm/sec CNT100;
   1:  PR[91,1] = PR[90,1] + -29.013;
   1:  PR[91,2] = PR[90,2] + -3.492;
   1:  PR[91,3] = PR[90,3] + 40.915;
   1:L PR[91] R[100]mm/sec CNT100;
   1:  PR[91,1] = PR[90,1] + -28.785;
   1:  PR[91,2] = PR[90,2] + -4.425;
   1:  PR[91,3] = PR[90,3] + 40.923;
   1:L PR[91] R[100]mm/sec CNT100;
   1:  PR[91,1] = PR[90,1] + -28.507;
   1:  PR[91,2] = PR[90,2] + -5.348;
   1:  PR[91,3] = PR[90,3] + 40.931;
   1:L PR[91] R[100]mm/sec CNT100;
   1:  PR[91,1] = PR[90,1] + -28.179;
   1:  PR[91,2] = PR[90,2] + -6.262;
   1:  PR[91,3] = PR[90,3] + 40.939;
   1:L PR[91] R[100]mm/sec CNT100;
   1:  PR[91,1] = PR[90,1] + -27.803;
   1:  PR[91,2] = PR[90,2] + -7.167;
   1:  PR[91,3] = PR[90,3] + 40.947;
   1:L PR[91] R[100]mm/sec CNT100;
   1:  PR[91,1] = PR[90,1] + -27.380;
   1:  PR[91,2] = PR[90,2] + -8.060;
   1:  PR[91,3] = PR[90,3] + 40.955;
   1:L PR[91] R[100]mm/sec CNT100;
   1:  PR[91,1] = PR[90,1] + -26.910;
   1:  PR[91,2] = PR[90,2] + -8.935;
   1:  PR[91,3] = PR[90,3] + 40.963;
   1:L PR[91] R[100]mm/sec CNT100;
   1:  PR[91,1] = PR[90,1] + -26.633;
   1:  PR[91,2] = PR[90,2] + -9.398;
   1:  PR[91,3] = PR[90,3] + 40.971;
   1:L PR[91] R[100]mm/sec CNT100;
   1:  PR[91,1] = PR[90,1] + -26.397;
   1:  PR[91,2] = PR[90,2] + -9.787;
   1:  PR[91,3] = PR[90,3] + 40.976;
   1:L PR[91] R[100]mm/sec CNT100;
   1:  PR[91,1] = PR[90,1] + -25.840;
   1:  PR[91,2] = PR[90,2] + -10.614;
   1:  PR[91,3] = PR[90,3] + 40.979;
   1:L PR[91] R[100]mm/sec CNT100;
   1:  PR[91,1] = PR[90,1] + -25.240;
   1:  PR[91,2] = PR[90,2] + -11.411;
   1:  PR[91,3] = PR[90,3] + 40.987;
   1:L PR[91] R[100]mm/sec CNT100;
   1:  PR[91,1] = PR[90,1] + -24.600;
   1:  PR[91,2] = PR[90,2] + -12.178;
   1:  PR[91,3] = PR[90,3] + 40.996;
   1:L PR[91] R[100]mm/sec CNT100;
   1:  PR[91,1] = PR[90,1] + -23.920;
   1:  PR[91,2] = PR[90,2] + -12.912;
   1:  PR[91,3] = PR[90,3] + 41.004;
   1:L PR[91] R[100]mm/sec CNT100;
   1:  PR[91,1] = PR[90,1] + -23.203;
   1:  PR[91,2] = PR[90,2] + -13.612;
   1:  PR[91,3] = PR[90,3] + 41.012;
   1:L PR[91] R[100]mm/sec CNT100;
   1:  PR[91,1] = PR[90,1] + -22.451;
   1:  PR[91,2] = PR[90,2] + -14.278;
   1:  PR[91,3] = PR[90,3] + 41.020;
   1:L PR[91] R[100]mm/sec CNT100;
   1:  PR[91,1] = PR[90,1] + -21.664;
   1:  PR[91,2] = PR[90,2] + -14.906;
   1:  PR[91,3] = PR[90,3] + 41.029;
   1:L PR[91] R[100]mm/sec CNT100;
   1:  PR[91,1] = PR[90,1] + -20.845;
   1:  PR[91,2] = PR[90,2] + -15.497;
   1:  PR[91,3] = PR[90,3] + 41.037;
   1:L PR[91] R[100]mm/sec CNT100;
   1:  PR[91,1] = PR[90,1] + -19.996;
   1:  PR[91,2] = PR[90,2] + -16.049;
   1:  PR[91,3] = PR[90,3] + 41.045;
   1:L PR[91] R[100]mm/sec CNT100;
   1:  PR[91,1] = PR[90,1] + -19.119;
   1:  PR[91,2] = PR[90,2] + -16.561;
   1:  PR[91,3] = PR[90,3] + 41.053;
   1:L PR[91] R[100]mm/sec CNT100;
   1:  PR[91,1] = PR[90,1] + -18.187;
   1:  PR[91,2] = PR[90,2] + -17.047;
   1:  PR[91,3] = PR[90,3] + 41.062;
   1:L PR[91] R[100]mm/sec CNT100;
   1:  PR[91,1] = PR[90,1] + -17.226;
   1:  PR[91,2] = PR[90,2] + -17.488;
   1:  PR[91,3] = PR[90,3] + 41.070;
   1:L PR[91] R[100]mm/sec CNT100;
   1:  PR[91,1] = PR[90,1] + -16.403;
   1:  PR[91,2] = PR[90,2] + -17.821;
   1:  PR[91,3] = PR[90,3] + 41.079;
   1:L PR[91] R[100]mm/sec CNT100;
   1:  PR[91,1] = PR[90,1] + -15.452;
   1:  PR[91,2] = PR[90,2] + -18.156;
   1:  PR[91,3] = PR[90,3] + 41.086;
   1:L PR[91] R[100]mm/sec CNT100;
   1:  PR[91,1] = PR[90,1] + -14.483;
   1:  PR[91,2] = PR[90,2] + -18.447;
   1:  PR[91,3] = PR[90,3] + 41.095;
   1:L PR[91] R[100]mm/sec CNT100;
   1:  PR[91,1] = PR[90,1] + -13.498;
   1:  PR[91,2] = PR[90,2] + -18.692;
   1:  PR[91,3] = PR[90,3] + 41.103;
   1:L PR[91] R[100]mm/sec CNT100;
   1:  PR[91,1] = PR[90,1] + -12.494;
   1:  PR[91,2] = PR[90,2] + -18.892;
   1:  PR[91,3] = PR[90,3] + 41.111;
   1:L PR[91] R[100]mm/sec CNT100;
   1:  PR[91,1] = PR[90,1] + -12.093;
   1:  PR[91,2] = PR[90,2] + -18.957;
   1:  PR[91,3] = PR[90,3] + 41.120;
   1:L PR[91] R[100]mm/sec CNT100;
   1:  PR[91,1] = PR[90,1] + -11.488;
   1:  PR[91,2] = PR[90,2] + -19.042;
   1:  PR[91,3] = PR[90,3] + 41.123;
   1:L PR[91] R[100]mm/sec CNT100;
   1:  PR[91,1] = PR[90,1] + -10.463;
   1:  PR[91,2] = PR[90,2] + -19.145;
   1:  PR[91,3] = PR[90,3] + 41.128;
   1:L PR[91] R[100]mm/sec CNT100;
   1:  PR[91,1] = PR[90,1] + -9.432;
   1:  PR[91,2] = PR[90,2] + -19.198;
   1:  PR[91,3] = PR[90,3] + 41.137;
   1:L PR[91] R[100]mm/sec CNT100;
   1:  PR[91,1] = PR[90,1] + -8.840;
   1:  PR[91,2] = PR[90,2] + -19.204;
   1:  PR[91,3] = PR[90,3] + 41.145;
   1:L PR[91] R[100]mm/sec CNT100;
   1:  PR[91,1] = PR[90,1] + -8.403;
   1:  PR[91,2] = PR[90,2] + -19.201;
   1:  PR[91,3] = PR[90,3] + 41.150;
   1:L PR[91] R[100]mm/sec CNT100;
   1:  PR[91,1] = PR[90,1] + -7.364;
   1:  PR[91,2] = PR[90,2] + -19.154;
   1:  PR[91,3] = PR[90,3] + 41.153;
   1:L PR[91] R[100]mm/sec CNT100;
   1:  PR[91,1] = PR[90,1] + -6.328;
   1:  PR[91,2] = PR[90,2] + -19.055;
   1:  PR[91,3] = PR[90,3] + 41.162;
   1:L PR[91] R[100]mm/sec CNT100;
   1:  PR[91,1] = PR[90,1] + -5.573;
   1:  PR[91,2] = PR[90,2] + -18.949;
   1:  PR[91,3] = PR[90,3] + 41.171;
   1:L PR[91] R[100]mm/sec CNT100;
   1:  PR[91,1] = PR[90,1] + -4.269;
   1:  PR[91,2] = PR[90,2] + -18.704;
   1:  PR[91,3] = PR[90,3] + 41.177;
   1:L PR[91] R[100]mm/sec CNT100;
   1:  PR[91,1] = PR[90,1] + -3.255;
   1:  PR[91,2] = PR[90,2] + -18.453;
   1:  PR[91,3] = PR[90,3] + 41.188;
   1:L PR[91] R[100]mm/sec CNT100;
   1:  PR[91,1] = PR[90,1] + -2.364;
   1:  PR[91,2] = PR[90,2] + -18.184;
   1:  PR[91,3] = PR[90,3] + 41.196;
   1:L PR[91] R[100]mm/sec CNT100;
   1:  PR[91,1] = PR[90,1] + -1.178;
   1:  PR[91,2] = PR[90,2] + -17.761;
   1:  PR[91,3] = PR[90,3] + 41.204;
   1:L PR[91] R[100]mm/sec CNT100;
   1:  PR[91,1] = PR[90,1] + -0.741;
   1:  PR[91,2] = PR[90,2] + -17.630;
   1:  PR[91,3] = PR[90,3] + 41.214;
   1:L PR[91] R[100]mm/sec CNT100;
   1:  PR[91,1] = PR[90,1] + -0.255;
   1:  PR[91,2] = PR[90,2] + -17.567;
   1:  PR[91,3] = PR[90,3] + 41.218;
   1:L PR[91] R[100]mm/sec CNT100;
   1:  PR[91,1] = PR[90,1] + 0.235;
   1:  PR[91,2] = PR[90,2] + -17.586;
   1:  PR[91,3] = PR[90,3] + 41.222;
   1:L PR[91] R[100]mm/sec CNT100;
   1:  PR[91,1] = PR[90,1] + 0.709;
   1:  PR[91,2] = PR[90,2] + -17.680;
   1:  PR[91,3] = PR[90,3] + 41.226;
   1:L PR[91] R[100]mm/sec CNT100;
   1:  PR[91] = PR[90];
   1:  PR[91,1] = PR[90,1] + 1.518;
   1:  PR[91,2] = PR[90,2] + -18.372;
   1:  PR[91,3] = PR[90,3] + 42.560;
   1:L PR[91] R[100]mm/sec CNT100;
   1:  PR[91,1] = PR[90,1] + 2.539;
   1:  PR[91,2] = PR[90,2] + -18.676;
   1:  PR[91,3] = PR[90,3] + 41.237;
   1:L PR[91] R[100]mm/sec CNT100;
   1:  PR[91,1] = PR[90,1] + 3.575;
   1:  PR[91,2] = PR[90,2] + -18.929;
   1:  PR[91,3] = PR[90,3] + 41.245;
   1:L PR[91] R[100]mm/sec CNT100;
   1:  PR[91,1] = PR[90,1] + 4.622;
   1:  PR[91,2] = PR[90,2] + -19.129;
   1:  PR[91,3] = PR[90,3] + 41.254;
   1:L PR[91] R[100]mm/sec CNT100;
   1:  PR[91,1] = PR[90,1] + 5.679;
   1:  PR[91,2] = PR[90,2] + -19.276;
   1:  PR[91,3] = PR[90,3] + 41.263;
   1:L PR[91] R[100]mm/sec CNT100;
   1:  PR[91,1] = PR[90,1] + 6.741;
   1:  PR[91,2] = PR[90,2] + -19.369;
   1:  PR[91,3] = PR[90,3] + 41.272;
   1:L PR[91] R[100]mm/sec CNT100;
   1:  PR[91,1] = PR[90,1] + 7.807;
   1:  PR[91,2] = PR[90,2] + -19.409;
   1:  PR[91,3] = PR[90,3] + 41.281;
   1:L PR[91] R[100]mm/sec CNT100;
   1:  PR[91,1] = PR[90,1] + 8.873;
   1:  PR[91,2] = PR[90,2] + -19.396;
   1:  PR[91,3] = PR[90,3] + 41.289;
   1:L PR[91] R[100]mm/sec CNT100;
   1:  PR[91,1] = PR[90,1] + 9.921;
   1:  PR[91,2] = PR[90,2] + -19.332;
   1:  PR[91,3] = PR[90,3] + 41.298;
   1:L PR[91] R[100]mm/sec CNT100;
   1:  PR[91,1] = PR[90,1] + 11.069;
   1:  PR[91,2] = PR[90,2] + -19.203;
   1:  PR[91,3] = PR[90,3] + 41.307;
   1:L PR[91] R[100]mm/sec CNT100;
   1:  PR[91,1] = PR[90,1] + 11.991;
   1:  PR[91,2] = PR[90,2] + -19.054;
   1:  PR[91,3] = PR[90,3] + 41.316;
   1:L PR[91] R[100]mm/sec CNT100;
   1:  PR[91,1] = PR[90,1] + 13.008;
   1:  PR[91,2] = PR[90,2] + -18.840;
   1:  PR[91,3] = PR[90,3] + 41.324;
   1:L PR[91] R[100]mm/sec CNT100;
   1:  PR[91,1] = PR[90,1] + 14.009;
   1:  PR[91,2] = PR[90,2] + -18.578;
   1:  PR[91,3] = PR[90,3] + 41.333;
   1:L PR[91] R[100]mm/sec CNT100;
   1:  PR[91,1] = PR[90,1] + 14.993;
   1:  PR[91,2] = PR[90,2] + -18.269;
   1:  PR[91,3] = PR[90,3] + 41.341;
   1:L PR[91] R[100]mm/sec CNT100;
   1:  PR[91,1] = PR[90,1] + 15.958;
   1:  PR[91,2] = PR[90,2] + -17.915;
   1:  PR[91,3] = PR[90,3] + 41.350;
   1:L PR[91] R[100]mm/sec CNT100;
   1:  PR[91,1] = PR[90,1] + 16.900;
   1:  PR[91,2] = PR[90,2] + -17.516;
   1:  PR[91,3] = PR[90,3] + 41.358;
   1:L PR[91] R[100]mm/sec CNT100;
   1:  PR[91,1] = PR[90,1] + 17.818;
   1:  PR[91,2] = PR[90,2] + -17.075;
   1:  PR[91,3] = PR[90,3] + 41.367;
   1:L PR[91] R[100]mm/sec CNT100;
   1:  PR[91,1] = PR[90,1] + 18.710;
   1:  PR[91,2] = PR[90,2] + -16.593;
   1:  PR[91,3] = PR[90,3] + 41.375;
   1:L PR[91] R[100]mm/sec CNT100;
   1:  PR[91,1] = PR[90,1] + 19.574;
   1:  PR[91,2] = PR[90,2] + -16.070;
   1:  PR[91,3] = PR[90,3] + 41.384;
   1:L PR[91] R[100]mm/sec CNT100;
   1:  PR[91,1] = PR[90,1] + 20.411;
   1:  PR[91,2] = PR[90,2] + -15.507;
   1:  PR[91,3] = PR[90,3] + 41.392;
   1:L PR[91] R[100]mm/sec CNT100;
   1:  PR[91,1] = PR[90,1] + 20.913;
   1:  PR[91,2] = PR[90,2] + -15.144;
   1:  PR[91,3] = PR[90,3] + 41.400;
   1:L PR[91] R[100]mm/sec CNT100;
   1:  PR[91,1] = PR[90,1] + 21.733;
   1:  PR[91,2] = PR[90,2] + -14.492;
   1:  PR[91,3] = PR[90,3] + 41.405;
   1:L PR[91] R[100]mm/sec CNT100;
   1:  PR[91,1] = PR[90,1] + 22.513;
   1:  PR[91,2] = PR[90,2] + -13.804;
   1:  PR[91,3] = PR[90,3] + 41.414;
   1:L PR[91] R[100]mm/sec CNT100;
   1:  PR[91,1] = PR[90,1] + 23.254;
   1:  PR[91,2] = PR[90,2] + -13.080;
   1:  PR[91,3] = PR[90,3] + 41.423;
   1:L PR[91] R[100]mm/sec CNT100;
   1:  PR[91,1] = PR[90,1] + 23.952;
   1:  PR[91,2] = PR[90,2] + -12.323;
   1:  PR[91,3] = PR[90,3] + 41.431;
   1:L PR[91] R[100]mm/sec CNT100;
   1:  PR[91,1] = PR[90,1] + 24.608;
   1:  PR[91,2] = PR[90,2] + -11.534;
   1:  PR[91,3] = PR[90,3] + 41.440;
   1:L PR[91] R[100]mm/sec CNT100;
   1:  PR[91,1] = PR[90,1] + 25.219;
   1:  PR[91,2] = PR[90,2] + -10.716;
   1:  PR[91,3] = PR[90,3] + 41.448;
   1:L PR[91] R[100]mm/sec CNT100;
   1:  PR[91,1] = PR[90,1] + 25.786;
   1:  PR[91,2] = PR[90,2] + -9.871;
   1:  PR[91,3] = PR[90,3] + 41.457;
   1:L PR[91] R[100]mm/sec CNT100;
   1:  PR[91,1] = PR[90,1] + 26.306;
   1:  PR[91,2] = PR[90,2] + -9.005;
   1:  PR[91,3] = PR[90,3] + 41.465;
   1:L PR[91] R[100]mm/sec CNT100;
   1:  PR[91,1] = PR[90,1] + 26.789;
   1:  PR[91,2] = PR[90,2] + -8.100;
   1:  PR[91,3] = PR[90,3] + 41.473;
   1:L PR[91] R[100]mm/sec CNT100;
   1:  PR[91,1] = PR[90,1] + 27.208;
   1:  PR[91,2] = PR[90,2] + -7.213;
   1:  PR[91,3] = PR[90,3] + 41.482;
   1:L PR[91] R[100]mm/sec CNT100;
   1:  PR[91,1] = PR[90,1] + 27.582;
   1:  PR[91,2] = PR[90,2] + -6.313;
   1:  PR[91,3] = PR[90,3] + 41.490;
   1:L PR[91] R[100]mm/sec CNT100;
   1:  PR[91,1] = PR[90,1] + 27.909;
   1:  PR[91,2] = PR[90,2] + -5.396;
   1:  PR[91,3] = PR[90,3] + 41.498;
   1:L PR[91] R[100]mm/sec CNT100;
   1:  PR[91,1] = PR[90,1] + 28.187;
   1:  PR[91,2] = PR[90,2] + -4.467;
   1:  PR[91,3] = PR[90,3] + 41.506;
   1:L PR[91] R[100]mm/sec CNT100;
   1:  PR[91,1] = PR[90,1] + 28.416;
   1:  PR[91,2] = PR[90,2] + -3.526;
   1:  PR[91,3] = PR[90,3] + 41.514;
   1:L PR[91] R[100]mm/sec CNT100;
   1:  PR[91,1] = PR[90,1] + 28.594;
   1:  PR[91,2] = PR[90,2] + -2.569;
   1:  PR[91,3] = PR[90,3] + 41.522;
   1:L PR[91] R[100]mm/sec CNT100;
   1:  PR[91,1] = PR[90,1] + 28.722;
   1:  PR[91,2] = PR[90,2] + -1.594;
   1:  PR[91,3] = PR[90,3] + 41.530;
   1:L PR[91] R[100]mm/sec CNT100;
   1:  PR[91,1] = PR[90,1] + 28.799;
   1:  PR[91,2] = PR[90,2] + -0.596;
   1:  PR[91,3] = PR[90,3] + 41.538;
   1:L PR[91] R[100]mm/sec CNT100;
   1:  PR[91,1] = PR[90,1] + 28.824;
   1:  PR[91,2] = PR[90,2] + 0.428;
   1:  PR[91,3] = PR[90,3] + 41.547;
   1:L PR[91] R[100]mm/sec CNT100;
   1:  PR[91,1] = PR[90,1] + 28.799;
   1:  PR[91,2] = PR[90,2] + 1.451;
   1:  PR[91,3] = PR[90,3] + 41.555;
   1:L PR[91] R[100]mm/sec CNT100;
   1:  PR[91,1] = PR[90,1] + 28.722;
   1:  PR[91,2] = PR[90,2] + 2.449;
   1:  PR[91,3] = PR[90,3] + 41.563;
   1:L PR[91] R[100]mm/sec CNT100;
   1:  PR[91,1] = PR[90,1] + 28.594;
   1:  PR[91,2] = PR[90,2] + 3.425;
   1:  PR[91,3] = PR[90,3] + 41.572;
   1:L PR[91] R[100]mm/sec CNT100;
   1:  PR[91,1] = PR[90,1] + 28.416;
   1:  PR[91,2] = PR[90,2] + 4.382;
   1:  PR[91,3] = PR[90,3] + 41.580;
   1:L PR[91] R[100]mm/sec CNT100;
   1:  PR[91,1] = PR[90,1] + 28.187;
   1:  PR[91,2] = PR[90,2] + 5.323;
   1:  PR[91,3] = PR[90,3] + 41.588;
   1:L PR[91] R[100]mm/sec CNT100;
   1:  PR[91,1] = PR[90,1] + 27.909;
   1:  PR[91,2] = PR[90,2] + 6.251;
   1:  PR[91,3] = PR[90,3] + 41.596;
   1:L PR[91] R[100]mm/sec CNT100;
   1:  PR[91,1] = PR[90,1] + 27.582;
   1:  PR[91,2] = PR[90,2] + 7.168;
   1:  PR[91,3] = PR[90,3] + 41.604;
   1:L PR[91] R[100]mm/sec CNT100;
   1:  PR[91,1] = PR[90,1] + 27.205;
   1:  PR[91,2] = PR[90,2] + 8.075;
   1:  PR[91,3] = PR[90,3] + 41.612;
   1:L PR[91] R[100]mm/sec CNT100;
   1:  PR[91,1] = PR[90,1] + 26.780;
   1:  PR[91,2] = PR[90,2] + 8.974;
   1:  PR[91,3] = PR[90,3] + 41.620;
   1:L PR[91] R[100]mm/sec CNT100;
   1:  PR[91,1] = PR[90,1] + 26.306;
   1:  PR[91,2] = PR[90,2] + 9.860;
   1:  PR[91,3] = PR[90,3] + 41.628;
   1:L PR[91] R[100]mm/sec CNT100;
   1:  PR[91,1] = PR[90,1] + 25.785;
   1:  PR[91,2] = PR[90,2] + 10.728;
   1:  PR[91,3] = PR[90,3] + 41.637;
   1:L PR[91] R[100]mm/sec CNT100;
   1:  PR[91,1] = PR[90,1] + 25.286;
   1:  PR[91,2] = PR[90,2] + 11.473;
   1:  PR[91,3] = PR[90,3] + 41.645;
   1:L PR[91] R[100]mm/sec CNT100;
   1:  PR[91,1] = PR[90,1] + 24.607;
   1:  PR[91,2] = PR[90,2] + 12.391;
   1:  PR[91,3] = PR[90,3] + 41.652;
   1:L PR[91] R[100]mm/sec CNT100;
   1:  PR[91,1] = PR[90,1] + 23.952;
   1:  PR[91,2] = PR[90,2] + 13.179;
   1:  PR[91,3] = PR[90,3] + 41.662;
   1:L PR[91] R[100]mm/sec CNT100;
   1:  PR[91,1] = PR[90,1] + 23.253;
   1:  PR[91,2] = PR[90,2] + 13.936;
   1:  PR[91,3] = PR[90,3] + 41.670;
   1:L PR[91] R[100]mm/sec CNT100;
   1:  PR[91,1] = PR[90,1] + 22.513;
   1:  PR[91,2] = PR[90,2] + 14.660;
   1:  PR[91,3] = PR[90,3] + 41.679;
   1:L PR[91] R[100]mm/sec CNT100;
   1:  PR[91,1] = PR[90,1] + 21.733;
   1:  PR[91,2] = PR[90,2] + 15.347;
   1:  PR[91,3] = PR[90,3] + 41.687;
   1:L PR[91] R[100]mm/sec CNT100;
   1:  PR[91,1] = PR[90,1] + 20.912;
   1:  PR[91,2] = PR[90,2] + 15.999;
   1:  PR[91,3] = PR[90,3] + 41.696;
   1:L PR[91] R[100]mm/sec CNT100;
   1:  PR[91,1] = PR[90,1] + 20.407;
   1:  PR[91,2] = PR[90,2] + 16.366;
   1:  PR[91,3] = PR[90,3] + 41.705;
   1:L PR[91] R[100]mm/sec CNT100;
   1:  PR[91,1] = PR[90,1] + 20.061;
   1:  PR[91,2] = PR[90,2] + 16.608;
   1:  PR[91,3] = PR[90,3] + 41.710;
   1:L PR[91] R[100]mm/sec CNT100;
   1:  PR[91,1] = PR[90,1] + 19.168;
   1:  PR[91,2] = PR[90,2] + 17.180;
   1:  PR[91,3] = PR[90,3] + 41.713;
   1:L PR[91] R[100]mm/sec CNT100;
   1:  PR[91,1] = PR[90,1] + 18.244;
   1:  PR[91,2] = PR[90,2] + 17.708;
   1:  PR[91,3] = PR[90,3] + 41.722;
   1:L PR[91] R[100]mm/sec CNT100;
   1:  PR[91,1] = PR[90,1] + 17.291;
   1:  PR[91,2] = PR[90,2] + 18.191;
   1:  PR[91,3] = PR[90,3] + 41.731;
   1:L PR[91] R[100]mm/sec CNT100;
   1:  PR[91,1] = PR[90,1] + 16.304;
   1:  PR[91,2] = PR[90,2] + 18.630;
   1:  PR[91,3] = PR[90,3] + 41.740;
   1:L PR[91] R[100]mm/sec CNT100;
   1:  PR[91,1] = PR[90,1] + 15.962;
   1:  PR[91,2] = PR[90,2] + 18.769;
   1:  PR[91,3] = PR[90,3] + 41.749;
   1:L PR[91] R[100]mm/sec CNT100;
   1:  PR[91,1] = PR[90,1] + 14.993;
   1:  PR[91,2] = PR[90,2] + 19.125;
   1:  PR[91,3] = PR[90,3] + 41.752;
   1:L PR[91] R[100]mm/sec CNT100;
   1:  PR[91,1] = PR[90,1] + 14.009;
   1:  PR[91,2] = PR[90,2] + 19.433;
   1:  PR[91,3] = PR[90,3] + 41.760;
   1:L PR[91] R[100]mm/sec CNT100;
   1:  PR[91,1] = PR[90,1] + 13.007;
   1:  PR[91,2] = PR[90,2] + 19.695;
   1:  PR[91,3] = PR[90,3] + 41.769;
   1:L PR[91] R[100]mm/sec CNT100;
   1:  PR[91,1] = PR[90,1] + 12.152;
   1:  PR[91,2] = PR[90,2] + 19.878;
   1:  PR[91,3] = PR[90,3] + 41.777;
   1:L PR[91] R[100]mm/sec CNT100;
   1:  PR[91,1] = PR[90,1] + 10.960;
   1:  PR[91,2] = PR[90,2] + 20.073;
   1:  PR[91,3] = PR[90,3] + 41.785;
   1:L PR[91] R[100]mm/sec CNT100;
   1:  PR[91,1] = PR[90,1] + 9.922;
   1:  PR[91,2] = PR[90,2] + 20.187;
   1:  PR[91,3] = PR[90,3] + 41.794;
   1:L PR[91] R[100]mm/sec CNT100;
   1:  PR[91,1] = PR[90,1] + 8.869;
   1:  PR[91,2] = PR[90,2] + 20.251;
   1:  PR[91,3] = PR[90,3] + 41.803;
   1:L PR[91] R[100]mm/sec CNT100;
   1:  PR[91,1] = PR[90,1] + 7.806;
   1:  PR[91,2] = PR[90,2] + 20.264;
   1:  PR[91,3] = PR[90,3] + 41.812;
   1:L PR[91] R[100]mm/sec CNT100;
   1:  PR[91,1] = PR[90,1] + 6.741;
   1:  PR[91,2] = PR[90,2] + 20.224;
   1:  PR[91,3] = PR[90,3] + 41.821;
   1:L PR[91] R[100]mm/sec CNT100;
   1:  PR[91,1] = PR[90,1] + 5.679;
   1:  PR[91,2] = PR[90,2] + 20.131;
   1:  PR[91,3] = PR[90,3] + 41.829;
   1:L PR[91] R[100]mm/sec CNT100;
   1:  PR[91,1] = PR[90,1] + 4.622;
   1:  PR[91,2] = PR[90,2] + 19.984;
   1:  PR[91,3] = PR[90,3] + 41.838;
   1:L PR[91] R[100]mm/sec CNT100;
   1:  PR[91,1] = PR[90,1] + 3.575;
   1:  PR[91,2] = PR[90,2] + 19.784;
   1:  PR[91,3] = PR[90,3] + 41.847;
   1:L PR[91] R[100]mm/sec CNT100;
   1:  PR[91,1] = PR[90,1] + 2.539;
   1:  PR[91,2] = PR[90,2] + 19.532;
   1:  PR[91,3] = PR[90,3] + 41.856;
   1:L PR[91] R[100]mm/sec CNT100;
   1:  PR[91,1] = PR[90,1] + 1.517;
   1:  PR[91,2] = PR[90,2] + 19.227;
   1:  PR[91,3] = PR[90,3] + 41.865;
   1:L PR[91] R[100]mm/sec CNT100;
   1:  PR[91,1] = PR[90,1] + 0.774;
   1:  PR[91,2] = PR[90,2] + 18.968;
   1:  PR[91,3] = PR[90,3] + 41.874;
   1:L PR[91] R[100]mm/sec CNT100;
   1:  PR[91,1] = PR[90,1] + 0.310;
   1:  PR[91,2] = PR[90,2] + 18.861;
   1:  PR[91,3] = PR[90,3] + 41.880;
   1:L PR[91] R[100]mm/sec CNT100;
   1:  PR[91,1] = PR[90,1] + -0.180;
   1:  PR[91,2] = PR[90,2] + 18.832;
   1:  PR[91,3] = PR[90,3] + 41.884;
   1:L PR[91] R[100]mm/sec CNT100;
   1:  PR[91,1] = PR[90,1] + -0.666;
   1:  PR[91,2] = PR[90,2] + 18.881;
   1:  PR[91,3] = PR[90,3] + 41.888;
   1:L PR[91] R[100]mm/sec CNT100;
   1:  PR[91,1] = PR[90,1] + -1.112;
   1:  PR[91,2] = PR[90,2] + 19.002;
   1:  PR[91,3] = PR[90,3] + 41.892;
   1:L PR[91] R[100]mm/sec CNT100;
   1:  PR[91,1] = PR[90,1] + -1.754;
   1:  PR[91,2] = PR[90,2] + 19.228;
   1:  PR[91,3] = PR[90,3] + 41.896;
   1:L PR[91] R[100]mm/sec CNT100;
   1:  PR[91,1] = PR[90,1] + -2.776;
   1:  PR[91,2] = PR[90,2] + 19.532;
   1:  PR[91,3] = PR[90,3] + 41.901;
   1:L PR[91] R[100]mm/sec CNT100;
   1:  PR[91,1] = PR[90,1] + -3.812;
   1:  PR[91,2] = PR[90,2] + 19.784;
   1:  PR[91,3] = PR[90,3] + 41.910;
   1:L PR[91] R[100]mm/sec CNT100;
   1:  PR[91,1] = PR[90,1] + -4.860;
   1:  PR[91,2] = PR[90,2] + 19.984;
   1:  PR[91,3] = PR[90,3] + 41.919;
   1:L PR[91] R[100]mm/sec CNT100;
   1:  PR[91,1] = PR[90,1] + -5.916;
   1:  PR[91,2] = PR[90,2] + 20.130;
   1:  PR[91,3] = PR[90,3] + 41.928;
   1:L PR[91] R[100]mm/sec CNT100;
   1:  PR[91,1] = PR[90,1] + -6.979;
   1:  PR[91,2] = PR[90,2] + 20.224;
   1:  PR[91,3] = PR[90,3] + 41.937;
   1:L PR[91] R[100]mm/sec CNT100;
   1:  PR[91,1] = PR[90,1] + -8.044;
   1:  PR[91,2] = PR[90,2] + 20.264;
   1:  PR[91,3] = PR[90,3] + 41.946;
   1:L PR[91] R[100]mm/sec CNT100;
   1:  PR[91,1] = PR[90,1] + -9.111;
   1:  PR[91,2] = PR[90,2] + 20.251;
   1:  PR[91,3] = PR[90,3] + 41.954;
   1:L PR[91] R[100]mm/sec CNT100;
   1:  PR[91,1] = PR[90,1] + -10.160;
   1:  PR[91,2] = PR[90,2] + 20.187;
   1:  PR[91,3] = PR[90,3] + 41.963;
   1:L PR[91] R[100]mm/sec CNT100;
   1:  PR[91,1] = PR[90,1] + -11.198;
   1:  PR[91,2] = PR[90,2] + 20.073;
   1:  PR[91,3] = PR[90,3] + 41.972;
   1:L PR[91] R[100]mm/sec CNT100;
   1:  PR[91,1] = PR[90,1] + -12.389;
   1:  PR[91,2] = PR[90,2] + 19.878;
   1:  PR[91,3] = PR[90,3] + 41.981;
   1:L PR[91] R[100]mm/sec CNT100;
   1:  PR[91,1] = PR[90,1] + -13.457;
   1:  PR[91,2] = PR[90,2] + 19.644;
   1:  PR[91,3] = PR[90,3] + 41.990;
   1:L PR[91] R[100]mm/sec CNT100;
   1:  PR[91,1] = PR[90,1] + -14.508;
   1:  PR[91,2] = PR[90,2] + 19.357;
   1:  PR[91,3] = PR[90,3] + 42.000;
   1:L PR[91] R[100]mm/sec CNT100;
   1:  PR[91,1] = PR[90,1] + -15.539;
   1:  PR[91,2] = PR[90,2] + 19.019;
   1:  PR[91,3] = PR[90,3] + 42.009;
   1:L PR[91] R[100]mm/sec CNT100;
   1:  PR[91,1] = PR[90,1] + -16.547;
   1:  PR[91,2] = PR[90,2] + 18.629;
   1:  PR[91,3] = PR[90,3] + 42.018;
   1:L PR[91] R[100]mm/sec CNT100;
   1:  PR[91,1] = PR[90,1] + -17.529;
   1:  PR[91,2] = PR[90,2] + 18.192;
   1:  PR[91,3] = PR[90,3] + 42.026;
   1:L PR[91] R[100]mm/sec CNT100;
   1:  PR[91,1] = PR[90,1] + -18.483;
   1:  PR[91,2] = PR[90,2] + 17.708;
   1:  PR[91,3] = PR[90,3] + 42.035;
   1:L PR[91] R[100]mm/sec CNT100;
   1:  PR[91,1] = PR[90,1] + -19.406;
   1:  PR[91,2] = PR[90,2] + 17.179;
   1:  PR[91,3] = PR[90,3] + 42.044;
   1:L PR[91] R[100]mm/sec CNT100;
   1:  PR[91,1] = PR[90,1] + -20.300;
   1:  PR[91,2] = PR[90,2] + 16.606;
   1:  PR[91,3] = PR[90,3] + 42.053;
   1:L PR[91] R[100]mm/sec CNT100;
   1:  PR[91,1] = PR[90,1] + -20.646;
   1:  PR[91,2] = PR[90,2] + 16.364;
   1:  PR[91,3] = PR[90,3] + 42.062;
   1:L PR[91] R[100]mm/sec CNT100;
   1:  PR[91,1] = PR[90,1] + -21.151;
   1:  PR[91,2] = PR[90,2] + 15.997;
   1:  PR[91,3] = PR[90,3] + 42.065;
   1:L PR[91] R[100]mm/sec CNT100;
   1:  PR[91,1] = PR[90,1] + -21.972;
   1:  PR[91,2] = PR[90,2] + 15.345;
   1:  PR[91,3] = PR[90,3] + 42.070;
   1:L PR[91] R[100]mm/sec CNT100;
   1:  PR[91,1] = PR[90,1] + -22.752;
   1:  PR[91,2] = PR[90,2] + 14.658;
   1:  PR[91,3] = PR[90,3] + 42.079;
   1:L PR[91] R[100]mm/sec CNT100;
   1:  PR[91,1] = PR[90,1] + -23.493;
   1:  PR[91,2] = PR[90,2] + 13.935;
   1:  PR[91,3] = PR[90,3] + 42.088;
   1:L PR[91] R[100]mm/sec CNT100;
   1:  PR[91,1] = PR[90,1] + -24.191;
   1:  PR[91,2] = PR[90,2] + 13.180;
   1:  PR[91,3] = PR[90,3] + 42.096;
   1:L PR[91] R[100]mm/sec CNT100;
   1:  PR[91,1] = PR[90,1] + -24.847;
   1:  PR[91,2] = PR[90,2] + 12.394;
   1:  PR[91,3] = PR[90,3] + 42.105;
   1:L PR[91] R[100]mm/sec CNT100;
   1:  PR[91,1] = PR[90,1] + -25.458;
   1:  PR[91,2] = PR[90,2] + 11.577;
   1:  PR[91,3] = PR[90,3] + 42.113;
   1:L PR[91] R[100]mm/sec CNT100;
   1:  PR[91,1] = PR[90,1] + -26.024;
   1:  PR[91,2] = PR[90,2] + 10.733;
   1:  PR[91,3] = PR[90,3] + 42.122;
   1:L PR[91] R[100]mm/sec CNT100;
   1:  PR[91,1] = PR[90,1] + -26.545;
   1:  PR[91,2] = PR[90,2] + 9.865;
   1:  PR[91,3] = PR[90,3] + 42.130;
   1:L PR[91] R[100]mm/sec CNT100;
   1:  PR[91,1] = PR[90,1] + -27.027;
   1:  PR[91,2] = PR[90,2] + 8.958;
   1:  PR[91,3] = PR[90,3] + 42.138;
   1:L PR[91] R[100]mm/sec CNT100;
   1:  PR[91,1] = PR[90,1] + -27.446;
   1:  PR[91,2] = PR[90,2] + 8.067;
   1:  PR[91,3] = PR[90,3] + 42.147;
   1:L PR[91] R[100]mm/sec CNT100;
   1:  PR[91,1] = PR[90,1] + -27.820;
   1:  PR[91,2] = PR[90,2] + 7.161;
   1:  PR[91,3] = PR[90,3] + 42.155;
   1:L PR[91] R[100]mm/sec CNT100;
   1:  PR[91,1] = PR[90,1] + -28.147;
   1:  PR[91,2] = PR[90,2] + 6.240;
   1:  PR[91,3] = PR[90,3] + 42.163;
   1:L PR[91] R[100]mm/sec CNT100;
   1:  PR[91,1] = PR[90,1] + -28.426;
   1:  PR[91,2] = PR[90,2] + 5.310;
   1:  PR[91,3] = PR[90,3] + 42.171;
   1:L PR[91] R[100]mm/sec CNT100;
   1:  PR[91,1] = PR[90,1] + -28.654;
   1:  PR[91,2] = PR[90,2] + 4.370;
   1:  PR[91,3] = PR[90,3] + 42.179;
   1:L PR[91] R[100]mm/sec CNT100;
   1:  PR[91,1] = PR[90,1] + -28.832;
   1:  PR[91,2] = PR[90,2] + 3.416;
   1:  PR[91,3] = PR[90,3] + 42.187;
   1:L PR[91] R[100]mm/sec CNT100;
   1:  PR[91,1] = PR[90,1] + -28.960;
   1:  PR[91,2] = PR[90,2] + 2.444;
   1:  PR[91,3] = PR[90,3] + 42.195;
   1:L PR[91] R[100]mm/sec CNT100;
   1:  PR[91,1] = PR[90,1] + -29.037;
   1:  PR[91,2] = PR[90,2] + 1.449;
   1:  PR[91,3] = PR[90,3] + 42.203;
   1:L PR[91] R[100]mm/sec CNT100;
   1:  PR[91,1] = PR[90,1] + -29.063;
   1:  PR[91,2] = PR[90,2] + 0.428;
   1:  PR[91,3] = PR[90,3] + 42.212;
   1:L PR[91] R[100]mm/sec CNT100;
   1:  PR[91,1] = PR[90,1] + -29.037;
   1:  PR[91,2] = PR[90,2] + -0.594;
   1:  PR[91,3] = PR[90,3] + 42.220;
   1:L PR[91] R[100]mm/sec CNT100;
   1:  PR[91,1] = PR[90,1] + -28.960;
   1:  PR[91,2] = PR[90,2] + -1.589;
   1:  PR[91,3] = PR[90,3] + 42.228;
   1:L PR[91] R[100]mm/sec CNT100;
   1:  PR[91,1] = PR[90,1] + -28.833;
   1:  PR[91,2] = PR[90,2] + -2.561;
   1:  PR[91,3] = PR[90,3] + 42.237;
   1:L PR[91] R[100]mm/sec CNT100;
   1:  PR[91,1] = PR[90,1] + -28.654;
   1:  PR[91,2] = PR[90,2] + -3.515;
   1:  PR[91,3] = PR[90,3] + 42.245;
   1:L PR[91] R[100]mm/sec CNT100;
   1:  PR[91,1] = PR[90,1] + -28.426;
   1:  PR[91,2] = PR[90,2] + -4.454;
   1:  PR[91,3] = PR[90,3] + 42.253;
   1:L PR[91] R[100]mm/sec CNT100;
   1:  PR[91,1] = PR[90,1] + -28.148;
   1:  PR[91,2] = PR[90,2] + -5.385;
   1:  PR[91,3] = PR[90,3] + 42.261;
   1:L PR[91] R[100]mm/sec CNT100;
   1:  PR[91,1] = PR[90,1] + -27.820;
   1:  PR[91,2] = PR[90,2] + -6.306;
   1:  PR[91,3] = PR[90,3] + 42.269;
   1:L PR[91] R[100]mm/sec CNT100;
   1:  PR[91,1] = PR[90,1] + -27.444;
   1:  PR[91,2] = PR[90,2] + -7.217;
   1:  PR[91,3] = PR[90,3] + 42.277;
   1:L PR[91] R[100]mm/sec CNT100;
   1:  PR[91,1] = PR[90,1] + -27.027;
   1:  PR[91,2] = PR[90,2] + -8.103;
   1:  PR[91,3] = PR[90,3] + 42.285;
   1:L PR[91] R[100]mm/sec CNT100;
   1:  PR[91,1] = PR[90,1] + -26.545;
   1:  PR[91,2] = PR[90,2] + -9.010;
   1:  PR[91,3] = PR[90,3] + 42.293;
   1:L PR[91] R[100]mm/sec CNT100;
   1:  PR[91,1] = PR[90,1] + -26.025;
   1:  PR[91,2] = PR[90,2] + -9.878;
   1:  PR[91,3] = PR[90,3] + 42.302;
   1:L PR[91] R[100]mm/sec CNT100;
   1:  PR[91,1] = PR[90,1] + -25.458;
   1:  PR[91,2] = PR[90,2] + -10.722;
   1:  PR[91,3] = PR[90,3] + 42.310;
   1:L PR[91] R[100]mm/sec CNT100;
   1:  PR[91,1] = PR[90,1] + -24.847;
   1:  PR[91,2] = PR[90,2] + -11.538;
   1:  PR[91,3] = PR[90,3] + 42.318;
   1:L PR[91] R[100]mm/sec CNT100;
   1:  PR[91,1] = PR[90,1] + -24.191;
   1:  PR[91,2] = PR[90,2] + -12.325;
   1:  PR[91,3] = PR[90,3] + 42.327;
   1:L PR[91] R[100]mm/sec CNT100;
   1:  PR[91,1] = PR[90,1] + -23.493;
   1:  PR[91,2] = PR[90,2] + -13.080;
   1:  PR[91,3] = PR[90,3] + 42.335;
   1:L PR[91] R[100]mm/sec CNT100;
   1:  PR[91,1] = PR[90,1] + -22.753;
   1:  PR[91,2] = PR[90,2] + -13.802;
   1:  PR[91,3] = PR[90,3] + 42.344;
   1:L PR[91] R[100]mm/sec CNT100;
   1:  PR[91,1] = PR[90,1] + -21.972;
   1:  PR[91,2] = PR[90,2] + -14.489;
   1:  PR[91,3] = PR[90,3] + 42.352;
   1:L PR[91] R[100]mm/sec CNT100;
   1:  PR[91,1] = PR[90,1] + -21.153;
   1:  PR[91,2] = PR[90,2] + -15.140;
   1:  PR[91,3] = PR[90,3] + 42.361;
   1:L PR[91] R[100]mm/sec CNT100;
   1:  PR[91,1] = PR[90,1] + -20.297;
   1:  PR[91,2] = PR[90,2] + -15.752;
   1:  PR[91,3] = PR[90,3] + 42.370;
   1:L PR[91] R[100]mm/sec CNT100;
   1:  PR[91,1] = PR[90,1] + -19.407;
   1:  PR[91,2] = PR[90,2] + -16.323;
   1:  PR[91,3] = PR[90,3] + 42.378;
   1:L PR[91] R[100]mm/sec CNT100;
   1:  PR[91,1] = PR[90,1] + -18.483;
   1:  PR[91,2] = PR[90,2] + -16.852;
   1:  PR[91,3] = PR[90,3] + 42.387;
   1:L PR[91] R[100]mm/sec CNT100;
   1:  PR[91,1] = PR[90,1] + -17.530;
   1:  PR[91,2] = PR[90,2] + -17.336;
   1:  PR[91,3] = PR[90,3] + 42.396;
   1:L PR[91] R[100]mm/sec CNT100;
   1:  PR[91,1] = PR[90,1] + -16.547;
   1:  PR[91,2] = PR[90,2] + -17.774;
   1:  PR[91,3] = PR[90,3] + 42.405;
   1:L PR[91] R[100]mm/sec CNT100;
   1:  PR[91,1] = PR[90,1] + -15.542;
   1:  PR[91,2] = PR[90,2] + -18.162;
   1:  PR[91,3] = PR[90,3] + 42.414;
   1:L PR[91] R[100]mm/sec CNT100;
   1:  PR[91,1] = PR[90,1] + -14.246;
   1:  PR[91,2] = PR[90,2] + -18.579;
   1:  PR[91,3] = PR[90,3] + 42.422;
   1:L PR[91] R[100]mm/sec CNT100;
   1:  PR[91,1] = PR[90,1] + -13.246;
   1:  PR[91,2] = PR[90,2] + -18.840;
   1:  PR[91,3] = PR[90,3] + 42.434;
   1:L PR[91] R[100]mm/sec CNT100;
   1:  PR[91,1] = PR[90,1] + -12.392;
   1:  PR[91,2] = PR[90,2] + -19.023;
   1:  PR[91,3] = PR[90,3] + 42.442;
   1:L PR[91] R[100]mm/sec CNT100;
   1:  PR[91,1] = PR[90,1] + -11.199;
   1:  PR[91,2] = PR[90,2] + -19.218;
   1:  PR[91,3] = PR[90,3] + 42.450;
   1:L PR[91] R[100]mm/sec CNT100;
   1:  PR[91,1] = PR[90,1] + -10.160;
   1:  PR[91,2] = PR[90,2] + -19.332;
   1:  PR[91,3] = PR[90,3] + 42.459;
   1:L PR[91] R[100]mm/sec CNT100;
   1:  PR[91,1] = PR[90,1] + -9.107;
   1:  PR[91,2] = PR[90,2] + -19.396;
   1:  PR[91,3] = PR[90,3] + 42.468;
   1:L PR[91] R[100]mm/sec CNT100;
   1:  PR[91,1] = PR[90,1] + -8.045;
   1:  PR[91,2] = PR[90,2] + -19.409;
   1:  PR[91,3] = PR[90,3] + 42.477;
   1:L PR[91] R[100]mm/sec CNT100;
   1:  PR[91,1] = PR[90,1] + -6.979;
   1:  PR[91,2] = PR[90,2] + -19.369;
   1:  PR[91,3] = PR[90,3] + 42.486;
   1:L PR[91] R[100]mm/sec CNT100;
   1:  PR[91,1] = PR[90,1] + -5.916;
   1:  PR[91,2] = PR[90,2] + -19.275;
   1:  PR[91,3] = PR[90,3] + 42.494;
   1:L PR[91] R[100]mm/sec CNT100;
   1:  PR[91,1] = PR[90,1] + -4.860;
   1:  PR[91,2] = PR[90,2] + -19.129;
   1:  PR[91,3] = PR[90,3] + 42.503;
   1:L PR[91] R[100]mm/sec CNT100;
   1:  PR[91,1] = PR[90,1] + -3.812;
   1:  PR[91,2] = PR[90,2] + -18.929;
   1:  PR[91,3] = PR[90,3] + 42.512;
   1:L PR[91] R[100]mm/sec CNT100;
   1:  PR[91,1] = PR[90,1] + -2.776;
   1:  PR[91,2] = PR[90,2] + -18.677;
   1:  PR[91,3] = PR[90,3] + 42.521;
   1:L PR[91] R[100]mm/sec CNT100;
   1:  PR[91,1] = PR[90,1] + -1.755;
   1:  PR[91,2] = PR[90,2] + -18.373;
   1:  PR[91,3] = PR[90,3] + 42.530;
   1:L PR[91] R[100]mm/sec CNT100;
   1:  PR[91,1] = PR[90,1] + -1.113;
   1:  PR[91,2] = PR[90,2] + -18.148;
   1:  PR[91,3] = PR[90,3] + 42.539;
   1:L PR[91] R[100]mm/sec CNT100;
   1:  PR[91,1] = PR[90,1] + -0.667;
   1:  PR[91,2] = PR[90,2] + -18.026;
   1:  PR[91,3] = PR[90,3] + 42.544;
   1:L PR[91] R[100]mm/sec CNT100;
   1:  PR[91,1] = PR[90,1] + -0.180;
   1:  PR[91,2] = PR[90,2] + -17.977;
   1:  PR[91,3] = PR[90,3] + 42.548;
   1:L PR[91] R[100]mm/sec CNT100;
   1:  PR[91,1] = PR[90,1] + 0.310;
   1:  PR[91,2] = PR[90,2] + -18.006;
   1:  PR[91,3] = PR[90,3] + 42.552;
   1:L PR[91] R[100]mm/sec CNT100;
   1:  PR[91,1] = PR[90,1] + 0.774;
   1:  PR[91,2] = PR[90,2] + -18.112;
   1:  PR[91,3] = PR[90,3] + 42.556;
   1:L PR[91] R[100]mm/sec CNT100;
   1:  PR[91] = PR[90];
   1:  PR[91,1] = PR[90,1] + 2.041;
   1:  PR[91,2] = PR[90,2] + -18.901;
   1:  PR[91,3] = PR[90,3] + 43.890;
   1:L PR[91] R[100]mm/sec CNT100;
   1:  PR[91,1] = PR[90,1] + 3.083;
   1:  PR[91,2] = PR[90,2] + -19.153;
   1:  PR[91,3] = PR[90,3] + 42.571;
   1:L PR[91] R[100]mm/sec CNT100;
   1:  PR[91,1] = PR[90,1] + 4.138;
   1:  PR[91,2] = PR[90,2] + -19.352;
   1:  PR[91,3] = PR[90,3] + 42.580;
   1:L PR[91] R[100]mm/sec CNT100;
   1:  PR[91,1] = PR[90,1] + 5.203;
   1:  PR[91,2] = PR[90,2] + -19.497;
   1:  PR[91,3] = PR[90,3] + 42.589;
   1:L PR[91] R[100]mm/sec CNT100;
   1:  PR[91,1] = PR[90,1] + 5.618;
   1:  PR[91,2] = PR[90,2] + -19.534;
   1:  PR[91,3] = PR[90,3] + 42.598;
   1:L PR[91] R[100]mm/sec CNT100;
   1:  PR[91,1] = PR[90,1] + 6.271;
   1:  PR[91,2] = PR[90,2] + -19.589;
   1:  PR[91,3] = PR[90,3] + 42.601;
   1:L PR[91] R[100]mm/sec CNT100;
   1:  PR[91,1] = PR[90,1] + 7.345;
   1:  PR[91,2] = PR[90,2] + -19.627;
   1:  PR[91,3] = PR[90,3] + 42.606;
   1:L PR[91] R[100]mm/sec CNT100;
   1:  PR[91,1] = PR[90,1] + 8.418;
   1:  PR[91,2] = PR[90,2] + -19.612;
   1:  PR[91,3] = PR[90,3] + 42.615;
   1:L PR[91] R[100]mm/sec CNT100;
   1:  PR[91,1] = PR[90,1] + 9.490;
   1:  PR[91,2] = PR[90,2] + -19.543;
   1:  PR[91,3] = PR[90,3] + 42.624;
   1:L PR[91] R[100]mm/sec CNT100;
   1:  PR[91,1] = PR[90,1] + 10.127;
   1:  PR[91,2] = PR[90,2] + -19.471;
   1:  PR[91,3] = PR[90,3] + 42.633;
   1:L PR[91] R[100]mm/sec CNT100;
   1:  PR[91,1] = PR[90,1] + 10.554;
   1:  PR[91,2] = PR[90,2] + -19.421;
   1:  PR[91,3] = PR[90,3] + 42.639;
   1:L PR[91] R[100]mm/sec CNT100;
   1:  PR[91,1] = PR[90,1] + 11.611;
   1:  PR[91,2] = PR[90,2] + -19.247;
   1:  PR[91,3] = PR[90,3] + 42.642;
   1:L PR[91] R[100]mm/sec CNT100;
   1:  PR[91,1] = PR[90,1] + 12.656;
   1:  PR[91,2] = PR[90,2] + -19.020;
   1:  PR[91,3] = PR[90,3] + 42.651;
   1:L PR[91] R[100]mm/sec CNT100;
   1:  PR[91,1] = PR[90,1] + 13.688;
   1:  PR[91,2] = PR[90,2] + -18.741;
   1:  PR[91,3] = PR[90,3] + 42.660;
   1:L PR[91] R[100]mm/sec CNT100;
   1:  PR[91,1] = PR[90,1] + 14.704;
   1:  PR[91,2] = PR[90,2] + -18.413;
   1:  PR[91,3] = PR[90,3] + 42.669;
   1:L PR[91] R[100]mm/sec CNT100;
   1:  PR[91,1] = PR[90,1] + 15.700;
   1:  PR[91,2] = PR[90,2] + -18.035;
   1:  PR[91,3] = PR[90,3] + 42.678;
   1:L PR[91] R[100]mm/sec CNT100;
   1:  PR[91,1] = PR[90,1] + 16.674;
   1:  PR[91,2] = PR[90,2] + -17.609;
   1:  PR[91,3] = PR[90,3] + 42.687;
   1:L PR[91] R[100]mm/sec CNT100;
   1:  PR[91,1] = PR[90,1] + 17.624;
   1:  PR[91,2] = PR[90,2] + -17.137;
   1:  PR[91,3] = PR[90,3] + 42.695;
   1:L PR[91] R[100]mm/sec CNT100;
   1:  PR[91,1] = PR[90,1] + 18.556;
   1:  PR[91,2] = PR[90,2] + -16.614;
   1:  PR[91,3] = PR[90,3] + 42.704;
   1:L PR[91] R[100]mm/sec CNT100;
   1:  PR[91,1] = PR[90,1] + 19.469;
   1:  PR[91,2] = PR[90,2] + -16.041;
   1:  PR[91,3] = PR[90,3] + 42.713;
   1:L PR[91] R[100]mm/sec CNT100;
   1:  PR[91,1] = PR[90,1] + 20.254;
   1:  PR[91,2] = PR[90,2] + -15.492;
   1:  PR[91,3] = PR[90,3] + 42.722;
   1:L PR[91] R[100]mm/sec CNT100;
   1:  PR[91,1] = PR[90,1] + 21.186;
   1:  PR[91,2] = PR[90,2] + -14.769;
   1:  PR[91,3] = PR[90,3] + 42.730;
   1:L PR[91] R[100]mm/sec CNT100;
   1:  PR[91,1] = PR[90,1] + 21.986;
   1:  PR[91,2] = PR[90,2] + -14.075;
   1:  PR[91,3] = PR[90,3] + 42.740;
   1:L PR[91] R[100]mm/sec CNT100;
   1:  PR[91,1] = PR[90,1] + 22.748;
   1:  PR[91,2] = PR[90,2] + -13.342;
   1:  PR[91,3] = PR[90,3] + 42.749;
   1:L PR[91] R[100]mm/sec CNT100;
   1:  PR[91,1] = PR[90,1] + 23.274;
   1:  PR[91,2] = PR[90,2] + -12.784;
   1:  PR[91,3] = PR[90,3] + 42.757;
   1:L PR[91] R[100]mm/sec CNT100;
   1:  PR[91,1] = PR[90,1] + 24.140;
   1:  PR[91,2] = PR[90,2] + -11.774;
   1:  PR[91,3] = PR[90,3] + 42.764;
   1:L PR[91] R[100]mm/sec CNT100;
   1:  PR[91,1] = PR[90,1] + 24.768;
   1:  PR[91,2] = PR[90,2] + -10.945;
   1:  PR[91,3] = PR[90,3] + 42.775;
   1:L PR[91] R[100]mm/sec CNT100;
   1:  PR[91,1] = PR[90,1] + 25.351;
   1:  PR[91,2] = PR[90,2] + -10.087;
   1:  PR[91,3] = PR[90,3] + 42.784;
   1:L PR[91] R[100]mm/sec CNT100;
   1:  PR[91,1] = PR[90,1] + 25.887;
   1:  PR[91,2] = PR[90,2] + -9.205;
   1:  PR[91,3] = PR[90,3] + 42.792;
   1:L PR[91] R[100]mm/sec CNT100;
   1:  PR[91,1] = PR[90,1] + 26.375;
   1:  PR[91,2] = PR[90,2] + -8.302;
   1:  PR[91,3] = PR[90,3] + 42.801;
   1:L PR[91] R[100]mm/sec CNT100;
   1:  PR[91,1] = PR[90,1] + 26.813;
   1:  PR[91,2] = PR[90,2] + -7.384;
   1:  PR[91,3] = PR[90,3] + 42.809;
   1:L PR[91] R[100]mm/sec CNT100;
   1:  PR[91,1] = PR[90,1] + 27.202;
   1:  PR[91,2] = PR[90,2] + -6.453;
   1:  PR[91,3] = PR[90,3] + 42.818;
   1:L PR[91] R[100]mm/sec CNT100;
   1:  PR[91,1] = PR[90,1] + 27.539;
   1:  PR[91,2] = PR[90,2] + -5.513;
   1:  PR[91,3] = PR[90,3] + 42.826;
   1:L PR[91] R[100]mm/sec CNT100;
   1:  PR[91,1] = PR[90,1] + 27.826;
   1:  PR[91,2] = PR[90,2] + -4.562;
   1:  PR[91,3] = PR[90,3] + 42.834;
   1:L PR[91] R[100]mm/sec CNT100;
   1:  PR[91,1] = PR[90,1] + 28.060;
   1:  PR[91,2] = PR[90,2] + -3.599;
   1:  PR[91,3] = PR[90,3] + 42.843;
   1:L PR[91] R[100]mm/sec CNT100;
   1:  PR[91,1] = PR[90,1] + 28.243;
   1:  PR[91,2] = PR[90,2] + -2.622;
   1:  PR[91,3] = PR[90,3] + 42.851;
   1:L PR[91] R[100]mm/sec CNT100;
   1:  PR[91,1] = PR[90,1] + 28.374;
   1:  PR[91,2] = PR[90,2] + -1.627;
   1:  PR[91,3] = PR[90,3] + 42.859;
   1:L PR[91] R[100]mm/sec CNT100;
   1:  PR[91,1] = PR[90,1] + 28.453;
   1:  PR[91,2] = PR[90,2] + -0.611;
   1:  PR[91,3] = PR[90,3] + 42.868;
   1:L PR[91] R[100]mm/sec CNT100;
   1:  PR[91,1] = PR[90,1] + 28.478;
   1:  PR[91,2] = PR[90,2] + 0.428;
   1:  PR[91,3] = PR[90,3] + 42.876;
   1:L PR[91] R[100]mm/sec CNT100;
   1:  PR[91,1] = PR[90,1] + 28.453;
   1:  PR[91,2] = PR[90,2] + 1.467;
   1:  PR[91,3] = PR[90,3] + 42.885;
   1:L PR[91] R[100]mm/sec CNT100;
   1:  PR[91,1] = PR[90,1] + 28.374;
   1:  PR[91,2] = PR[90,2] + 2.482;
   1:  PR[91,3] = PR[90,3] + 42.893;
   1:L PR[91] R[100]mm/sec CNT100;
   1:  PR[91,1] = PR[90,1] + 28.243;
   1:  PR[91,2] = PR[90,2] + 3.477;
   1:  PR[91,3] = PR[90,3] + 42.902;
   1:L PR[91] R[100]mm/sec CNT100;
   1:  PR[91,1] = PR[90,1] + 28.060;
   1:  PR[91,2] = PR[90,2] + 4.454;
   1:  PR[91,3] = PR[90,3] + 42.910;
   1:L PR[91] R[100]mm/sec CNT100;
   1:  PR[91,1] = PR[90,1] + 27.825;
   1:  PR[91,2] = PR[90,2] + 5.417;
   1:  PR[91,3] = PR[90,3] + 42.918;
   1:L PR[91] R[100]mm/sec CNT100;
   1:  PR[91,1] = PR[90,1] + 27.539;
   1:  PR[91,2] = PR[90,2] + 6.368;
   1:  PR[91,3] = PR[90,3] + 42.927;
   1:L PR[91] R[100]mm/sec CNT100;
   1:  PR[91,1] = PR[90,1] + 27.201;
   1:  PR[91,2] = PR[90,2] + 7.309;
   1:  PR[91,3] = PR[90,3] + 42.935;
   1:L PR[91] R[100]mm/sec CNT100;
   1:  PR[91,1] = PR[90,1] + 27.019;
   1:  PR[91,2] = PR[90,2] + 7.751;
   1:  PR[91,3] = PR[90,3] + 42.943;
   1:L PR[91] R[100]mm/sec CNT100;
   1:  PR[91,1] = PR[90,1] + 26.814;
   1:  PR[91,2] = PR[90,2] + 8.238;
   1:  PR[91,3] = PR[90,3] + 42.947;
   1:L PR[91] R[100]mm/sec CNT100;
   1:  PR[91,1] = PR[90,1] + 26.375;
   1:  PR[91,2] = PR[90,2] + 9.158;
   1:  PR[91,3] = PR[90,3] + 42.952;
   1:L PR[91] R[100]mm/sec CNT100;
   1:  PR[91,1] = PR[90,1] + 25.887;
   1:  PR[91,2] = PR[90,2] + 10.060;
   1:  PR[91,3] = PR[90,3] + 42.960;
   1:L PR[91] R[100]mm/sec CNT100;
   1:  PR[91,1] = PR[90,1] + 25.351;
   1:  PR[91,2] = PR[90,2] + 10.943;
   1:  PR[91,3] = PR[90,3] + 42.969;
   1:L PR[91] R[100]mm/sec CNT100;
   1:  PR[91,1] = PR[90,1] + 24.766;
   1:  PR[91,2] = PR[90,2] + 11.803;
   1:  PR[91,3] = PR[90,3] + 42.977;
   1:L PR[91] R[100]mm/sec CNT100;
   1:  PR[91,1] = PR[90,1] + 24.561;
   1:  PR[91,2] = PR[90,2] + 12.078;
   1:  PR[91,3] = PR[90,3] + 42.986;
   1:L PR[91] R[100]mm/sec CNT100;
   1:  PR[91,1] = PR[90,1] + 24.139;
   1:  PR[91,2] = PR[90,2] + 12.631;
   1:  PR[91,3] = PR[90,3] + 42.989;
   1:L PR[91] R[100]mm/sec CNT100;
   1:  PR[91,1] = PR[90,1] + 23.464;
   1:  PR[91,2] = PR[90,2] + 13.431;
   1:  PR[91,3] = PR[90,3] + 42.995;
   1:L PR[91] R[100]mm/sec CNT100;
   1:  PR[91,1] = PR[90,1] + 22.746;
   1:  PR[91,2] = PR[90,2] + 14.199;
   1:  PR[91,3] = PR[90,3] + 43.003;
   1:L PR[91] R[100]mm/sec CNT100;
   1:  PR[91,1] = PR[90,1] + 21.986;
   1:  PR[91,2] = PR[90,2] + 14.930;
   1:  PR[91,3] = PR[90,3] + 43.012;
   1:L PR[91] R[100]mm/sec CNT100;
   1:  PR[91,1] = PR[90,1] + 21.185;
   1:  PR[91,2] = PR[90,2] + 15.625;
   1:  PR[91,3] = PR[90,3] + 43.021;
   1:L PR[91] R[100]mm/sec CNT100;
   1:  PR[91,1] = PR[90,1] + 20.346;
   1:  PR[91,2] = PR[90,2] + 16.281;
   1:  PR[91,3] = PR[90,3] + 43.030;
   1:L PR[91] R[100]mm/sec CNT100;
   1:  PR[91,1] = PR[90,1] + 19.412;
   1:  PR[91,2] = PR[90,2] + 16.933;
   1:  PR[91,3] = PR[90,3] + 43.038;
   1:L PR[91] R[100]mm/sec CNT100;
   1:  PR[91,1] = PR[90,1] + 18.539;
   1:  PR[91,2] = PR[90,2] + 17.479;
   1:  PR[91,3] = PR[90,3] + 43.048;
   1:L PR[91] R[100]mm/sec CNT100;
   1:  PR[91,1] = PR[90,1] + 17.624;
   1:  PR[91,2] = PR[90,2] + 17.992;
   1:  PR[91,3] = PR[90,3] + 43.056;
   1:L PR[91] R[100]mm/sec CNT100;
   1:  PR[91,1] = PR[90,1] + 16.674;
   1:  PR[91,2] = PR[90,2] + 18.464;
   1:  PR[91,3] = PR[90,3] + 43.065;
   1:L PR[91] R[100]mm/sec CNT100;
   1:  PR[91,1] = PR[90,1] + 15.700;
   1:  PR[91,2] = PR[90,2] + 18.890;
   1:  PR[91,3] = PR[90,3] + 43.074;
   1:L PR[91] R[100]mm/sec CNT100;
   1:  PR[91,1] = PR[90,1] + 14.704;
   1:  PR[91,2] = PR[90,2] + 19.268;
   1:  PR[91,3] = PR[90,3] + 43.083;
   1:L PR[91] R[100]mm/sec CNT100;
   1:  PR[91,1] = PR[90,1] + 13.688;
   1:  PR[91,2] = PR[90,2] + 19.597;
   1:  PR[91,3] = PR[90,3] + 43.092;
   1:L PR[91] R[100]mm/sec CNT100;
   1:  PR[91,1] = PR[90,1] + 12.657;
   1:  PR[91,2] = PR[90,2] + 19.875;
   1:  PR[91,3] = PR[90,3] + 43.101;
   1:L PR[91] R[100]mm/sec CNT100;
   1:  PR[91,1] = PR[90,1] + 11.611;
   1:  PR[91,2] = PR[90,2] + 20.102;
   1:  PR[91,3] = PR[90,3] + 43.109;
   1:L PR[91] R[100]mm/sec CNT100;
   1:  PR[91,1] = PR[90,1] + 10.554;
   1:  PR[91,2] = PR[90,2] + 20.277;
   1:  PR[91,3] = PR[90,3] + 43.118;
   1:L PR[91] R[100]mm/sec CNT100;
   1:  PR[91,1] = PR[90,1] + 10.128;
   1:  PR[91,2] = PR[90,2] + 20.326;
   1:  PR[91,3] = PR[90,3] + 43.127;
   1:L PR[91] R[100]mm/sec CNT100;
   1:  PR[91,1] = PR[90,1] + 9.490;
   1:  PR[91,2] = PR[90,2] + 20.398;
   1:  PR[91,3] = PR[90,3] + 43.131;
   1:L PR[91] R[100]mm/sec CNT100;
   1:  PR[91,1] = PR[90,1] + 8.419;
   1:  PR[91,2] = PR[90,2] + 20.467;
   1:  PR[91,3] = PR[90,3] + 43.136;
   1:L PR[91] R[100]mm/sec CNT100;
   1:  PR[91,1] = PR[90,1] + 7.346;
   1:  PR[91,2] = PR[90,2] + 20.483;
   1:  PR[91,3] = PR[90,3] + 43.145;
   1:L PR[91] R[100]mm/sec CNT100;
   1:  PR[91,1] = PR[90,1] + 6.273;
   1:  PR[91,2] = PR[90,2] + 20.444;
   1:  PR[91,3] = PR[90,3] + 43.154;
   1:L PR[91] R[100]mm/sec CNT100;
   1:  PR[91,1] = PR[90,1] + 5.203;
   1:  PR[91,2] = PR[90,2] + 20.353;
   1:  PR[91,3] = PR[90,3] + 43.163;
   1:L PR[91] R[100]mm/sec CNT100;
   1:  PR[91,1] = PR[90,1] + 4.139;
   1:  PR[91,2] = PR[90,2] + 20.207;
   1:  PR[91,3] = PR[90,3] + 43.172;
   1:L PR[91] R[100]mm/sec CNT100;
   1:  PR[91,1] = PR[90,1] + 3.084;
   1:  PR[91,2] = PR[90,2] + 20.008;
   1:  PR[91,3] = PR[90,3] + 43.181;
   1:L PR[91] R[100]mm/sec CNT100;
   1:  PR[91,1] = PR[90,1] + 2.043;
   1:  PR[91,2] = PR[90,2] + 19.757;
   1:  PR[91,3] = PR[90,3] + 43.190;
   1:L PR[91] R[100]mm/sec CNT100;
   1:  PR[91,1] = PR[90,1] + 0.802;
   1:  PR[91,2] = PR[90,2] + 19.381;
   1:  PR[91,3] = PR[90,3] + 43.199;
   1:L PR[91] R[100]mm/sec CNT100;
   1:  PR[91,1] = PR[90,1] + 0.383;
   1:  PR[91,2] = PR[90,2] + 19.275;
   1:  PR[91,3] = PR[90,3] + 43.209;
   1:L PR[91] R[100]mm/sec CNT100;
   1:  PR[91,1] = PR[90,1] + -0.105;
   1:  PR[91,2] = PR[90,2] + 19.233;
   1:  PR[91,3] = PR[90,3] + 43.213;
   1:L PR[91] R[100]mm/sec CNT100;
   1:  PR[91,1] = PR[90,1] + -0.591;
   1:  PR[91,2] = PR[90,2] + 19.271;
   1:  PR[91,3] = PR[90,3] + 43.217;
   1:L PR[91] R[100]mm/sec CNT100;
   1:  PR[91,1] = PR[90,1] + -0.907;
   1:  PR[91,2] = PR[90,2] + 19.345;
   1:  PR[91,3] = PR[90,3] + 43.221;
   1:L PR[91] R[100]mm/sec CNT100;
   1:  PR[91,1] = PR[90,1] + -2.278;
   1:  PR[91,2] = PR[90,2] + 19.757;
   1:  PR[91,3] = PR[90,3] + 43.224;
   1:L PR[91] R[100]mm/sec CNT100;
   1:  PR[91,1] = PR[90,1] + -3.321;
   1:  PR[91,2] = PR[90,2] + 20.008;
   1:  PR[91,3] = PR[90,3] + 43.236;
   1:L PR[91] R[100]mm/sec CNT100;
   1:  PR[91,1] = PR[90,1] + -4.376;
   1:  PR[91,2] = PR[90,2] + 20.207;
   1:  PR[91,3] = PR[90,3] + 43.245;
   1:L PR[91] R[100]mm/sec CNT100;
   1:  PR[91,1] = PR[90,1] + -5.440;
   1:  PR[91,2] = PR[90,2] + 20.352;
   1:  PR[91,3] = PR[90,3] + 43.254;
   1:L PR[91] R[100]mm/sec CNT100;
   1:  PR[91,1] = PR[90,1] + -6.510;
   1:  PR[91,2] = PR[90,2] + 20.444;
   1:  PR[91,3] = PR[90,3] + 43.263;
   1:L PR[91] R[100]mm/sec CNT100;
   1:  PR[91,1] = PR[90,1] + -7.584;
   1:  PR[91,2] = PR[90,2] + 20.482;
   1:  PR[91,3] = PR[90,3] + 43.271;
   1:L PR[91] R[100]mm/sec CNT100;
   1:  PR[91,1] = PR[90,1] + -8.111;
   1:  PR[91,2] = PR[90,2] + 20.476;
   1:  PR[91,3] = PR[90,3] + 43.280;
   1:L PR[91] R[100]mm/sec CNT100;
   1:  PR[91,1] = PR[90,1] + -8.656;
   1:  PR[91,2] = PR[90,2] + 20.467;
   1:  PR[91,3] = PR[90,3] + 43.285;
   1:L PR[91] R[100]mm/sec CNT100;
   1:  PR[91,1] = PR[90,1] + -9.727;
   1:  PR[91,2] = PR[90,2] + 20.398;
   1:  PR[91,3] = PR[90,3] + 43.289;
   1:L PR[91] R[100]mm/sec CNT100;
   1:  PR[91,1] = PR[90,1] + -10.792;
   1:  PR[91,2] = PR[90,2] + 20.276;
   1:  PR[91,3] = PR[90,3] + 43.298;
   1:L PR[91] R[100]mm/sec CNT100;
   1:  PR[91,1] = PR[90,1] + -11.849;
   1:  PR[91,2] = PR[90,2] + 20.102;
   1:  PR[91,3] = PR[90,3] + 43.307;
   1:L PR[91] R[100]mm/sec CNT100;
   1:  PR[91,1] = PR[90,1] + -12.895;
   1:  PR[91,2] = PR[90,2] + 19.875;
   1:  PR[91,3] = PR[90,3] + 43.316;
   1:L PR[91] R[100]mm/sec CNT100;
   1:  PR[91,1] = PR[90,1] + -13.926;
   1:  PR[91,2] = PR[90,2] + 19.598;
   1:  PR[91,3] = PR[90,3] + 43.325;
   1:L PR[91] R[100]mm/sec CNT100;
   1:  PR[91,1] = PR[90,1] + -14.942;
   1:  PR[91,2] = PR[90,2] + 19.269;
   1:  PR[91,3] = PR[90,3] + 43.334;
   1:L PR[91] R[100]mm/sec CNT100;
   1:  PR[91,1] = PR[90,1] + -15.937;
   1:  PR[91,2] = PR[90,2] + 18.891;
   1:  PR[91,3] = PR[90,3] + 43.343;
   1:L PR[91] R[100]mm/sec CNT100;
   1:  PR[91,1] = PR[90,1] + -16.912;
   1:  PR[91,2] = PR[90,2] + 18.465;
   1:  PR[91,3] = PR[90,3] + 43.352;
   1:L PR[91] R[100]mm/sec CNT100;
   1:  PR[91,1] = PR[90,1] + -17.862;
   1:  PR[91,2] = PR[90,2] + 17.992;
   1:  PR[91,3] = PR[90,3] + 43.360;
   1:L PR[91] R[100]mm/sec CNT100;
   1:  PR[91,1] = PR[90,1] + -18.793;
   1:  PR[91,2] = PR[90,2] + 17.469;
   1:  PR[91,3] = PR[90,3] + 43.369;
   1:L PR[91] R[100]mm/sec CNT100;
   1:  PR[91,1] = PR[90,1] + -19.706;
   1:  PR[91,2] = PR[90,2] + 16.895;
   1:  PR[91,3] = PR[90,3] + 43.378;
   1:L PR[91] R[100]mm/sec CNT100;
   1:  PR[91,1] = PR[90,1] + -20.584;
   1:  PR[91,2] = PR[90,2] + 16.279;
   1:  PR[91,3] = PR[90,3] + 43.387;
   1:L PR[91] R[100]mm/sec CNT100;
   1:  PR[91,1] = PR[90,1] + -21.300;
   1:  PR[91,2] = PR[90,2] + 15.723;
   1:  PR[91,3] = PR[90,3] + 43.396;
   1:L PR[91] R[100]mm/sec CNT100;
   1:  PR[91,1] = PR[90,1] + -22.226;
   1:  PR[91,2] = PR[90,2] + 14.928;
   1:  PR[91,3] = PR[90,3] + 43.404;
   1:L PR[91] R[100]mm/sec CNT100;
   1:  PR[91,1] = PR[90,1] + -22.985;
   1:  PR[91,2] = PR[90,2] + 14.198;
   1:  PR[91,3] = PR[90,3] + 43.414;
   1:L PR[91] R[100]mm/sec CNT100;
   1:  PR[91,1] = PR[90,1] + -23.703;
   1:  PR[91,2] = PR[90,2] + 13.433;
   1:  PR[91,3] = PR[90,3] + 43.422;
   1:L PR[91] R[100]mm/sec CNT100;
   1:  PR[91,1] = PR[90,1] + -24.378;
   1:  PR[91,2] = PR[90,2] + 12.635;
   1:  PR[91,3] = PR[90,3] + 43.431;
   1:L PR[91] R[100]mm/sec CNT100;
   1:  PR[91,1] = PR[90,1] + -25.007;
   1:  PR[91,2] = PR[90,2] + 11.806;
   1:  PR[91,3] = PR[90,3] + 43.440;
   1:L PR[91] R[100]mm/sec CNT100;
   1:  PR[91,1] = PR[90,1] + -25.589;
   1:  PR[91,2] = PR[90,2] + 10.948;
   1:  PR[91,3] = PR[90,3] + 43.449;
   1:L PR[91] R[100]mm/sec CNT100;
   1:  PR[91,1] = PR[90,1] + -26.125;
   1:  PR[91,2] = PR[90,2] + 10.065;
   1:  PR[91,3] = PR[90,3] + 43.457;
   1:L PR[91] R[100]mm/sec CNT100;
   1:  PR[91,1] = PR[90,1] + -26.613;
   1:  PR[91,2] = PR[90,2] + 9.160;
   1:  PR[91,3] = PR[90,3] + 43.466;
   1:L PR[91] R[100]mm/sec CNT100;
   1:  PR[91,1] = PR[90,1] + -27.051;
   1:  PR[91,2] = PR[90,2] + 8.238;
   1:  PR[91,3] = PR[90,3] + 43.474;
   1:L PR[91] R[100]mm/sec CNT100;
   1:  PR[91,1] = PR[90,1] + -27.440;
   1:  PR[91,2] = PR[90,2] + 7.302;
   1:  PR[91,3] = PR[90,3] + 43.483;
   1:L PR[91] R[100]mm/sec CNT100;
   1:  PR[91,1] = PR[90,1] + -27.612;
   1:  PR[91,2] = PR[90,2] + 6.825;
   1:  PR[91,3] = PR[90,3] + 43.491;
   1:L PR[91] R[100]mm/sec CNT100;
   1:  PR[91,1] = PR[90,1] + -27.777;
   1:  PR[91,2] = PR[90,2] + 6.359;
   1:  PR[91,3] = PR[90,3] + 43.495;
   1:L PR[91] R[100]mm/sec CNT100;
   1:  PR[91,1] = PR[90,1] + -28.064;
   1:  PR[91,2] = PR[90,2] + 5.405;
   1:  PR[91,3] = PR[90,3] + 43.500;
   1:L PR[91] R[100]mm/sec CNT100;
   1:  PR[91,1] = PR[90,1] + -28.299;
   1:  PR[91,2] = PR[90,2] + 4.443;
   1:  PR[91,3] = PR[90,3] + 43.508;
   1:L PR[91] R[100]mm/sec CNT100;
   1:  PR[91,1] = PR[90,1] + -28.482;
   1:  PR[91,2] = PR[90,2] + 3.469;
   1:  PR[91,3] = PR[90,3] + 43.516;
   1:L PR[91] R[100]mm/sec CNT100;
   1:  PR[91,1] = PR[90,1] + -28.613;
   1:  PR[91,2] = PR[90,2] + 2.478;
   1:  PR[91,3] = PR[90,3] + 43.524;
   1:L PR[91] R[100]mm/sec CNT100;
   1:  PR[91,1] = PR[90,1] + -28.691;
   1:  PR[91,2] = PR[90,2] + 1.466;
   1:  PR[91,3] = PR[90,3] + 43.533;
   1:L PR[91] R[100]mm/sec CNT100;
   1:  PR[91,1] = PR[90,1] + -28.717;
   1:  PR[91,2] = PR[90,2] + 0.428;
   1:  PR[91,3] = PR[90,3] + 43.541;
   1:L PR[91] R[100]mm/sec CNT100;
   1:  PR[91,1] = PR[90,1] + -28.691;
   1:  PR[91,2] = PR[90,2] + -0.610;
   1:  PR[91,3] = PR[90,3] + 43.550;
   1:L PR[91] R[100]mm/sec CNT100;
   1:  PR[91,1] = PR[90,1] + -28.613;
   1:  PR[91,2] = PR[90,2] + -1.623;
   1:  PR[91,3] = PR[90,3] + 43.558;
   1:L PR[91] R[100]mm/sec CNT100;
   1:  PR[91,1] = PR[90,1] + -28.482;
   1:  PR[91,2] = PR[90,2] + -2.614;
   1:  PR[91,3] = PR[90,3] + 43.567;
   1:L PR[91] R[100]mm/sec CNT100;
   1:  PR[91,1] = PR[90,1] + -28.299;
   1:  PR[91,2] = PR[90,2] + -3.588;
   1:  PR[91,3] = PR[90,3] + 43.575;
   1:L PR[91] R[100]mm/sec CNT100;
   1:  PR[91,1] = PR[90,1] + -28.064;
   1:  PR[91,2] = PR[90,2] + -4.550;
   1:  PR[91,3] = PR[90,3] + 43.583;
   1:L PR[91] R[100]mm/sec CNT100;
   1:  PR[91,1] = PR[90,1] + -27.778;
   1:  PR[91,2] = PR[90,2] + -5.504;
   1:  PR[91,3] = PR[90,3] + 43.592;
   1:L PR[91] R[100]mm/sec CNT100;
   1:  PR[91,1] = PR[90,1] + -27.612;
   1:  PR[91,2] = PR[90,2] + -5.971;
   1:  PR[91,3] = PR[90,3] + 43.600;
   1:L PR[91] R[100]mm/sec CNT100;
   1:  PR[91,1] = PR[90,1] + -27.440;
   1:  PR[91,2] = PR[90,2] + -6.447;
   1:  PR[91,3] = PR[90,3] + 43.604;
   1:L PR[91] R[100]mm/sec CNT100;
   1:  PR[91,1] = PR[90,1] + -27.051;
   1:  PR[91,2] = PR[90,2] + -7.382;
   1:  PR[91,3] = PR[90,3] + 43.608;
   1:L PR[91] R[100]mm/sec CNT100;
   1:  PR[91,1] = PR[90,1] + -26.612;
   1:  PR[91,2] = PR[90,2] + -8.306;
   1:  PR[91,3] = PR[90,3] + 43.617;
   1:L PR[91] R[100]mm/sec CNT100;
   1:  PR[91,1] = PR[90,1] + -26.408;
   1:  PR[91,2] = PR[90,2] + -8.689;
   1:  PR[91,3] = PR[90,3] + 43.625;
   1:L PR[91] R[100]mm/sec CNT100;
   1:  PR[91,1] = PR[90,1] + -26.126;
   1:  PR[91,2] = PR[90,2] + -9.209;
   1:  PR[91,3] = PR[90,3] + 43.629;
   1:L PR[91] R[100]mm/sec CNT100;
   1:  PR[91,1] = PR[90,1] + -25.590;
   1:  PR[91,2] = PR[90,2] + -10.093;
   1:  PR[91,3] = PR[90,3] + 43.634;
   1:L PR[91] R[100]mm/sec CNT100;
   1:  PR[91,1] = PR[90,1] + -25.007;
   1:  PR[91,2] = PR[90,2] + -10.951;
   1:  PR[91,3] = PR[90,3] + 43.642;
   1:L PR[91] R[100]mm/sec CNT100;
   1:  PR[91,1] = PR[90,1] + -24.378;
   1:  PR[91,2] = PR[90,2] + -11.780;
   1:  PR[91,3] = PR[90,3] + 43.651;
   1:L PR[91] R[100]mm/sec CNT100;
   1:  PR[91,1] = PR[90,1] + -23.704;
   1:  PR[91,2] = PR[90,2] + -12.578;
   1:  PR[91,3] = PR[90,3] + 43.660;
   1:L PR[91] R[100]mm/sec CNT100;
   1:  PR[91,1] = PR[90,1] + -22.986;
   1:  PR[91,2] = PR[90,2] + -13.343;
   1:  PR[91,3] = PR[90,3] + 43.668;
   1:L PR[91] R[100]mm/sec CNT100;
   1:  PR[91,1] = PR[90,1] + -22.225;
   1:  PR[91,2] = PR[90,2] + -14.074;
   1:  PR[91,3] = PR[90,3] + 43.677;
   1:L PR[91] R[100]mm/sec CNT100;
   1:  PR[91,1] = PR[90,1] + -21.424;
   1:  PR[91,2] = PR[90,2] + -14.768;
   1:  PR[91,3] = PR[90,3] + 43.686;
   1:L PR[91] R[100]mm/sec CNT100;
   1:  PR[91,1] = PR[90,1] + -20.584;
   1:  PR[91,2] = PR[90,2] + -15.424;
   1:  PR[91,3] = PR[90,3] + 43.695;
   1:L PR[91] R[100]mm/sec CNT100;
   1:  PR[91,1] = PR[90,1] + -19.706;
   1:  PR[91,2] = PR[90,2] + -16.040;
   1:  PR[91,3] = PR[90,3] + 43.703;
   1:L PR[91] R[100]mm/sec CNT100;
   1:  PR[91,1] = PR[90,1] + -18.777;
   1:  PR[91,2] = PR[90,2] + -16.623;
   1:  PR[91,3] = PR[90,3] + 43.712;
   1:L PR[91] R[100]mm/sec CNT100;
   1:  PR[91,1] = PR[90,1] + -17.862;
   1:  PR[91,2] = PR[90,2] + -17.137;
   1:  PR[91,3] = PR[90,3] + 43.721;
   1:L PR[91] R[100]mm/sec CNT100;
   1:  PR[91,1] = PR[90,1] + -16.912;
   1:  PR[91,2] = PR[90,2] + -17.610;
   1:  PR[91,3] = PR[90,3] + 43.730;
   1:L PR[91] R[100]mm/sec CNT100;
   1:  PR[91,1] = PR[90,1] + -15.938;
   1:  PR[91,2] = PR[90,2] + -18.036;
   1:  PR[91,3] = PR[90,3] + 43.739;
   1:L PR[91] R[100]mm/sec CNT100;
   1:  PR[91,1] = PR[90,1] + -14.942;
   1:  PR[91,2] = PR[90,2] + -18.414;
   1:  PR[91,3] = PR[90,3] + 43.748;
   1:L PR[91] R[100]mm/sec CNT100;
   1:  PR[91,1] = PR[90,1] + -13.926;
   1:  PR[91,2] = PR[90,2] + -18.743;
   1:  PR[91,3] = PR[90,3] + 43.757;
   1:L PR[91] R[100]mm/sec CNT100;
   1:  PR[91,1] = PR[90,1] + -12.895;
   1:  PR[91,2] = PR[90,2] + -19.020;
   1:  PR[91,3] = PR[90,3] + 43.766;
   1:L PR[91] R[100]mm/sec CNT100;
   1:  PR[91,1] = PR[90,1] + -11.849;
   1:  PR[91,2] = PR[90,2] + -19.247;
   1:  PR[91,3] = PR[90,3] + 43.774;
   1:L PR[91] R[100]mm/sec CNT100;
   1:  PR[91,1] = PR[90,1] + -10.792;
   1:  PR[91,2] = PR[90,2] + -19.421;
   1:  PR[91,3] = PR[90,3] + 43.783;
   1:L PR[91] R[100]mm/sec CNT100;
   1:  PR[91,1] = PR[90,1] + -9.727;
   1:  PR[91,2] = PR[90,2] + -19.543;
   1:  PR[91,3] = PR[90,3] + 43.792;
   1:L PR[91] R[100]mm/sec CNT100;
   1:  PR[91,1] = PR[90,1] + -8.655;
   1:  PR[91,2] = PR[90,2] + -19.612;
   1:  PR[91,3] = PR[90,3] + 43.801;
   1:L PR[91] R[100]mm/sec CNT100;
   1:  PR[91,1] = PR[90,1] + -8.110;
   1:  PR[91,2] = PR[90,2] + -19.621;
   1:  PR[91,3] = PR[90,3] + 43.810;
   1:L PR[91] R[100]mm/sec CNT100;
   1:  PR[91,1] = PR[90,1] + -7.583;
   1:  PR[91,2] = PR[90,2] + -19.627;
   1:  PR[91,3] = PR[90,3] + 43.815;
   1:L PR[91] R[100]mm/sec CNT100;
   1:  PR[91,1] = PR[90,1] + -6.509;
   1:  PR[91,2] = PR[90,2] + -19.589;
   1:  PR[91,3] = PR[90,3] + 43.819;
   1:L PR[91] R[100]mm/sec CNT100;
   1:  PR[91,1] = PR[90,1] + -5.439;
   1:  PR[91,2] = PR[90,2] + -19.497;
   1:  PR[91,3] = PR[90,3] + 43.828;
   1:L PR[91] R[100]mm/sec CNT100;
   1:  PR[91,1] = PR[90,1] + -4.375;
   1:  PR[91,2] = PR[90,2] + -19.351;
   1:  PR[91,3] = PR[90,3] + 43.837;
   1:L PR[91] R[100]mm/sec CNT100;
   1:  PR[91,1] = PR[90,1] + -3.319;
   1:  PR[91,2] = PR[90,2] + -19.153;
   1:  PR[91,3] = PR[90,3] + 43.846;
   1:L PR[91] R[100]mm/sec CNT100;
   1:  PR[91,1] = PR[90,1] + -2.278;
   1:  PR[91,2] = PR[90,2] + -18.901;
   1:  PR[91,3] = PR[90,3] + 43.855;
   1:L PR[91] R[100]mm/sec CNT100;
   1:  PR[91,1] = PR[90,1] + -1.037;
   1:  PR[91,2] = PR[90,2] + -18.526;
   1:  PR[91,3] = PR[90,3] + 43.864;
   1:L PR[91] R[100]mm/sec CNT100;
   1:  PR[91,1] = PR[90,1] + -0.594;
   1:  PR[91,2] = PR[90,2] + -18.416;
   1:  PR[91,3] = PR[90,3] + 43.874;
   1:L PR[91] R[100]mm/sec CNT100;
   1:  PR[91,1] = PR[90,1] + -0.105;
   1:  PR[91,2] = PR[90,2] + -18.378;
   1:  PR[91,3] = PR[90,3] + 43.878;
   1:L PR[91] R[100]mm/sec CNT100;
   1:  PR[91,1] = PR[90,1] + 0.383;
   1:  PR[91,2] = PR[90,2] + -18.420;
   1:  PR[91,3] = PR[90,3] + 43.882;
   1:L PR[91] R[100]mm/sec CNT100;
   1:  PR[91,1] = PR[90,1] + 0.802;
   1:  PR[91,2] = PR[90,2] + -18.526;
   1:  PR[91,3] = PR[90,3] + 43.886;
   1:L PR[91] R[100]mm/sec CNT100;
   1:  PR[91] = PR[90];
   1:  PR[91,1] = PR[90,1] + 1.522;
   1:  PR[91,2] = PR[90,2] + -19.127;
   1:  PR[91,3] = PR[90,3] + 45.220;
   1:L PR[91] R[100]mm/sec CNT100;
   1:  PR[91,1] = PR[90,1] + 2.580;
   1:  PR[91,2] = PR[90,2] + -19.380;
   1:  PR[91,3] = PR[90,3] + 43.899;
   1:L PR[91] R[100]mm/sec CNT100;
   1:  PR[91,1] = PR[90,1] + 3.645;
   1:  PR[91,2] = PR[90,2] + -19.578;
   1:  PR[91,3] = PR[90,3] + 43.908;
   1:L PR[91] R[100]mm/sec CNT100;
   1:  PR[91,1] = PR[90,1] + 4.720;
   1:  PR[91,2] = PR[90,2] + -19.722;
   1:  PR[91,3] = PR[90,3] + 43.917;
   1:L PR[91] R[100]mm/sec CNT100;
   1:  PR[91,1] = PR[90,1] + 5.800;
   1:  PR[91,2] = PR[90,2] + -19.811;
   1:  PR[91,3] = PR[90,3] + 43.926;
   1:L PR[91] R[100]mm/sec CNT100;
   1:  PR[91,1] = PR[90,1] + 6.883;
   1:  PR[91,2] = PR[90,2] + -19.846;
   1:  PR[91,3] = PR[90,3] + 43.936;
   1:L PR[91] R[100]mm/sec CNT100;
   1:  PR[91,1] = PR[90,1] + 7.964;
   1:  PR[91,2] = PR[90,2] + -19.828;
   1:  PR[91,3] = PR[90,3] + 43.945;
   1:L PR[91] R[100]mm/sec CNT100;
   1:  PR[91,1] = PR[90,1] + 9.042;
   1:  PR[91,2] = PR[90,2] + -19.757;
   1:  PR[91,3] = PR[90,3] + 43.954;
   1:L PR[91] R[100]mm/sec CNT100;
   1:  PR[91,1] = PR[90,1] + 10.114;
   1:  PR[91,2] = PR[90,2] + -19.632;
   1:  PR[91,3] = PR[90,3] + 43.963;
   1:L PR[91] R[100]mm/sec CNT100;
   1:  PR[91,1] = PR[90,1] + 11.178;
   1:  PR[91,2] = PR[90,2] + -19.454;
   1:  PR[91,3] = PR[90,3] + 43.972;
   1:L PR[91] R[100]mm/sec CNT100;
   1:  PR[91,1] = PR[90,1] + 12.230;
   1:  PR[91,2] = PR[90,2] + -19.224;
   1:  PR[91,3] = PR[90,3] + 43.981;
   1:L PR[91] R[100]mm/sec CNT100;
   1:  PR[91,1] = PR[90,1] + 13.269;
   1:  PR[91,2] = PR[90,2] + -18.941;
   1:  PR[91,3] = PR[90,3] + 43.990;
   1:L PR[91] R[100]mm/sec CNT100;
   1:  PR[91,1] = PR[90,1] + 14.291;
   1:  PR[91,2] = PR[90,2] + -18.608;
   1:  PR[91,3] = PR[90,3] + 43.999;
   1:L PR[91] R[100]mm/sec CNT100;
   1:  PR[91,1] = PR[90,1] + 15.293;
   1:  PR[91,2] = PR[90,2] + -18.226;
   1:  PR[91,3] = PR[90,3] + 44.008;
   1:L PR[91] R[100]mm/sec CNT100;
   1:  PR[91,1] = PR[90,1] + 16.274;
   1:  PR[91,2] = PR[90,2] + -17.795;
   1:  PR[91,3] = PR[90,3] + 44.017;
   1:L PR[91] R[100]mm/sec CNT100;
   1:  PR[91,1] = PR[90,1] + 17.230;
   1:  PR[91,2] = PR[90,2] + -17.317;
   1:  PR[91,3] = PR[90,3] + 44.026;
   1:L PR[91] R[100]mm/sec CNT100;
   1:  PR[91,1] = PR[90,1] + 18.159;
   1:  PR[91,2] = PR[90,2] + -16.793;
   1:  PR[91,3] = PR[90,3] + 44.035;
   1:L PR[91] R[100]mm/sec CNT100;
   1:  PR[91,1] = PR[90,1] + 19.058;
   1:  PR[91,2] = PR[90,2] + -16.225;
   1:  PR[91,3] = PR[90,3] + 44.044;
   1:L PR[91] R[100]mm/sec CNT100;
   1:  PR[91,1] = PR[90,1] + 19.563;
   1:  PR[91,2] = PR[90,2] + -15.871;
   1:  PR[91,3] = PR[90,3] + 44.052;
   1:L PR[91] R[100]mm/sec CNT100;
   1:  PR[91,1] = PR[90,1] + 19.925;
   1:  PR[91,2] = PR[90,2] + -15.615;
   1:  PR[91,3] = PR[90,3] + 44.058;
   1:L PR[91] R[100]mm/sec CNT100;
   1:  PR[91,1] = PR[90,1] + 20.759;
   1:  PR[91,2] = PR[90,2] + -14.963;
   1:  PR[91,3] = PR[90,3] + 44.061;
   1:L PR[91] R[100]mm/sec CNT100;
   1:  PR[91,1] = PR[90,1] + 21.557;
   1:  PR[91,2] = PR[90,2] + -14.271;
   1:  PR[91,3] = PR[90,3] + 44.070;
   1:L PR[91] R[100]mm/sec CNT100;
   1:  PR[91,1] = PR[90,1] + 22.317;
   1:  PR[91,2] = PR[90,2] + -13.541;
   1:  PR[91,3] = PR[90,3] + 44.079;
   1:L PR[91] R[100]mm/sec CNT100;
   1:  PR[91,1] = PR[90,1] + 23.037;
   1:  PR[91,2] = PR[90,2] + -12.774;
   1:  PR[91,3] = PR[90,3] + 44.088;
   1:L PR[91] R[100]mm/sec CNT100;
   1:  PR[91,1] = PR[90,1] + 23.715;
   1:  PR[91,2] = PR[90,2] + -11.973;
   1:  PR[91,3] = PR[90,3] + 44.097;
   1:L PR[91] R[100]mm/sec CNT100;
   1:  PR[91,1] = PR[90,1] + 24.349;
   1:  PR[91,2] = PR[90,2] + -11.139;
   1:  PR[91,3] = PR[90,3] + 44.105;
   1:L PR[91] R[100]mm/sec CNT100;
   1:  PR[91,1] = PR[90,1] + 24.939;
   1:  PR[91,2] = PR[90,2] + -10.275;
   1:  PR[91,3] = PR[90,3] + 44.114;
   1:L PR[91] R[100]mm/sec CNT100;
   1:  PR[91,1] = PR[90,1] + 25.483;
   1:  PR[91,2] = PR[90,2] + -9.385;
   1:  PR[91,3] = PR[90,3] + 44.123;
   1:L PR[91] R[100]mm/sec CNT100;
   1:  PR[91,1] = PR[90,1] + 25.979;
   1:  PR[91,2] = PR[90,2] + -8.472;
   1:  PR[91,3] = PR[90,3] + 44.132;
   1:L PR[91] R[100]mm/sec CNT100;
   1:  PR[91,1] = PR[90,1] + 26.427;
   1:  PR[91,2] = PR[90,2] + -7.540;
   1:  PR[91,3] = PR[90,3] + 44.140;
   1:L PR[91] R[100]mm/sec CNT100;
   1:  PR[91,1] = PR[90,1] + 26.824;
   1:  PR[91,2] = PR[90,2] + -6.594;
   1:  PR[91,3] = PR[90,3] + 44.149;
   1:L PR[91] R[100]mm/sec CNT100;
   1:  PR[91,1] = PR[90,1] + 27.170;
   1:  PR[91,2] = PR[90,2] + -5.636;
   1:  PR[91,3] = PR[90,3] + 44.158;
   1:L PR[91] R[100]mm/sec CNT100;
   1:  PR[91,1] = PR[90,1] + 27.464;
   1:  PR[91,2] = PR[90,2] + -4.665;
   1:  PR[91,3] = PR[90,3] + 44.166;
   1:L PR[91] R[100]mm/sec CNT100;
   1:  PR[91,1] = PR[90,1] + 27.705;
   1:  PR[91,2] = PR[90,2] + -3.681;
   1:  PR[91,3] = PR[90,3] + 44.175;
   1:L PR[91] R[100]mm/sec CNT100;
   1:  PR[91,1] = PR[90,1] + 27.894;
   1:  PR[91,2] = PR[90,2] + -2.682;
   1:  PR[91,3] = PR[90,3] + 44.183;
   1:L PR[91] R[100]mm/sec CNT100;
   1:  PR[91,1] = PR[90,1] + 28.029;
   1:  PR[91,2] = PR[90,2] + -1.666;
   1:  PR[91,3] = PR[90,3] + 44.192;
   1:L PR[91] R[100]mm/sec CNT100;
   1:  PR[91,1] = PR[90,1] + 28.110;
   1:  PR[91,2] = PR[90,2] + -0.630;
   1:  PR[91,3] = PR[90,3] + 44.200;
   1:L PR[91] R[100]mm/sec CNT100;
   1:  PR[91,1] = PR[90,1] + 28.137;
   1:  PR[91,2] = PR[90,2] + 0.428;
   1:  PR[91,3] = PR[90,3] + 44.209;
   1:L PR[91] R[100]mm/sec CNT100;
   1:  PR[91,1] = PR[90,1] + 28.110;
   1:  PR[91,2] = PR[90,2] + 1.485;
   1:  PR[91,3] = PR[90,3] + 44.218;
   1:L PR[91] R[100]mm/sec CNT100;
   1:  PR[91,1] = PR[90,1] + 28.029;
   1:  PR[91,2] = PR[90,2] + 2.521;
   1:  PR[91,3] = PR[90,3] + 44.227;
   1:L PR[91] R[100]mm/sec CNT100;
   1:  PR[91,1] = PR[90,1] + 27.894;
   1:  PR[91,2] = PR[90,2] + 3.537;
   1:  PR[91,3] = PR[90,3] + 44.235;
   1:L PR[91] R[100]mm/sec CNT100;
   1:  PR[91,1] = PR[90,1] + 27.703;
   1:  PR[91,2] = PR[90,2] + 4.548;
   1:  PR[91,3] = PR[90,3] + 44.244;
   1:L PR[91] R[100]mm/sec CNT100;
   1:  PR[91,1] = PR[90,1] + 27.463;
   1:  PR[91,2] = PR[90,2] + 5.522;
   1:  PR[91,3] = PR[90,3] + 44.252;
   1:L PR[91] R[100]mm/sec CNT100;
   1:  PR[91,1] = PR[90,1] + 27.163;
   1:  PR[91,2] = PR[90,2] + 6.509;
   1:  PR[91,3] = PR[90,3] + 44.261;
   1:L PR[91] R[100]mm/sec CNT100;
   1:  PR[91,1] = PR[90,1] + 26.824;
   1:  PR[91,2] = PR[90,2] + 7.450;
   1:  PR[91,3] = PR[90,3] + 44.269;
   1:L PR[91] R[100]mm/sec CNT100;
   1:  PR[91,1] = PR[90,1] + 26.427;
   1:  PR[91,2] = PR[90,2] + 8.395;
   1:  PR[91,3] = PR[90,3] + 44.278;
   1:L PR[91] R[100]mm/sec CNT100;
   1:  PR[91,1] = PR[90,1] + 25.979;
   1:  PR[91,2] = PR[90,2] + 9.327;
   1:  PR[91,3] = PR[90,3] + 44.286;
   1:L PR[91] R[100]mm/sec CNT100;
   1:  PR[91,1] = PR[90,1] + 25.483;
   1:  PR[91,2] = PR[90,2] + 10.240;
   1:  PR[91,3] = PR[90,3] + 44.295;
   1:L PR[91] R[100]mm/sec CNT100;
   1:  PR[91,1] = PR[90,1] + 24.939;
   1:  PR[91,2] = PR[90,2] + 11.130;
   1:  PR[91,3] = PR[90,3] + 44.304;
   1:L PR[91] R[100]mm/sec CNT100;
   1:  PR[91,1] = PR[90,1] + 24.349;
   1:  PR[91,2] = PR[90,2] + 11.994;
   1:  PR[91,3] = PR[90,3] + 44.312;
   1:L PR[91] R[100]mm/sec CNT100;
   1:  PR[91,1] = PR[90,1] + 23.715;
   1:  PR[91,2] = PR[90,2] + 12.828;
   1:  PR[91,3] = PR[90,3] + 44.321;
   1:L PR[91] R[100]mm/sec CNT100;
   1:  PR[91,1] = PR[90,1] + 23.037;
   1:  PR[91,2] = PR[90,2] + 13.629;
   1:  PR[91,3] = PR[90,3] + 44.330;
   1:L PR[91] R[100]mm/sec CNT100;
   1:  PR[91,1] = PR[90,1] + 22.317;
   1:  PR[91,2] = PR[90,2] + 14.396;
   1:  PR[91,3] = PR[90,3] + 44.339;
   1:L PR[91] R[100]mm/sec CNT100;
   1:  PR[91,1] = PR[90,1] + 21.557;
   1:  PR[91,2] = PR[90,2] + 15.126;
   1:  PR[91,3] = PR[90,3] + 44.348;
   1:L PR[91] R[100]mm/sec CNT100;
   1:  PR[91,1] = PR[90,1] + 20.760;
   1:  PR[91,2] = PR[90,2] + 15.818;
   1:  PR[91,3] = PR[90,3] + 44.356;
   1:L PR[91] R[100]mm/sec CNT100;
   1:  PR[91,1] = PR[90,1] + 19.925;
   1:  PR[91,2] = PR[90,2] + 16.470;
   1:  PR[91,3] = PR[90,3] + 44.365;
   1:L PR[91] R[100]mm/sec CNT100;
   1:  PR[91,1] = PR[90,1] + 19.564;
   1:  PR[91,2] = PR[90,2] + 16.726;
   1:  PR[91,3] = PR[90,3] + 44.374;
   1:L PR[91] R[100]mm/sec CNT100;
   1:  PR[91,1] = PR[90,1] + 19.059;
   1:  PR[91,2] = PR[90,2] + 17.080;
   1:  PR[91,3] = PR[90,3] + 44.378;
   1:L PR[91] R[100]mm/sec CNT100;
   1:  PR[91,1] = PR[90,1] + 18.159;
   1:  PR[91,2] = PR[90,2] + 17.648;
   1:  PR[91,3] = PR[90,3] + 44.383;
   1:L PR[91] R[100]mm/sec CNT100;
   1:  PR[91,1] = PR[90,1] + 17.230;
   1:  PR[91,2] = PR[90,2] + 18.172;
   1:  PR[91,3] = PR[90,3] + 44.392;
   1:L PR[91] R[100]mm/sec CNT100;
   1:  PR[91,1] = PR[90,1] + 16.274;
   1:  PR[91,2] = PR[90,2] + 18.650;
   1:  PR[91,3] = PR[90,3] + 44.401;
   1:L PR[91] R[100]mm/sec CNT100;
   1:  PR[91,1] = PR[90,1] + 15.294;
   1:  PR[91,2] = PR[90,2] + 19.081;
   1:  PR[91,3] = PR[90,3] + 44.410;
   1:L PR[91] R[100]mm/sec CNT100;
   1:  PR[91,1] = PR[90,1] + 14.291;
   1:  PR[91,2] = PR[90,2] + 19.463;
   1:  PR[91,3] = PR[90,3] + 44.419;
   1:L PR[91] R[100]mm/sec CNT100;
   1:  PR[91,1] = PR[90,1] + 13.270;
   1:  PR[91,2] = PR[90,2] + 19.796;
   1:  PR[91,3] = PR[90,3] + 44.428;
   1:L PR[91] R[100]mm/sec CNT100;
   1:  PR[91,1] = PR[90,1] + 12.231;
   1:  PR[91,2] = PR[90,2] + 20.079;
   1:  PR[91,3] = PR[90,3] + 44.437;
   1:L PR[91] R[100]mm/sec CNT100;
   1:  PR[91,1] = PR[90,1] + 11.179;
   1:  PR[91,2] = PR[90,2] + 20.309;
   1:  PR[91,3] = PR[90,3] + 44.446;
   1:L PR[91] R[100]mm/sec CNT100;
   1:  PR[91,1] = PR[90,1] + 10.116;
   1:  PR[91,2] = PR[90,2] + 20.487;
   1:  PR[91,3] = PR[90,3] + 44.455;
   1:L PR[91] R[100]mm/sec CNT100;
   1:  PR[91,1] = PR[90,1] + 9.043;
   1:  PR[91,2] = PR[90,2] + 20.612;
   1:  PR[91,3] = PR[90,3] + 44.464;
   1:L PR[91] R[100]mm/sec CNT100;
   1:  PR[91,1] = PR[90,1] + 7.966;
   1:  PR[91,2] = PR[90,2] + 20.684;
   1:  PR[91,3] = PR[90,3] + 44.473;
   1:L PR[91] R[100]mm/sec CNT100;
   1:  PR[91,1] = PR[90,1] + 6.880;
   1:  PR[91,2] = PR[90,2] + 20.701;
   1:  PR[91,3] = PR[90,3] + 44.482;
   1:L PR[91] R[100]mm/sec CNT100;
   1:  PR[91,1] = PR[90,1] + 5.801;
   1:  PR[91,2] = PR[90,2] + 20.666;
   1:  PR[91,3] = PR[90,3] + 44.491;
   1:L PR[91] R[100]mm/sec CNT100;
   1:  PR[91,1] = PR[90,1] + 4.722;
   1:  PR[91,2] = PR[90,2] + 20.577;
   1:  PR[91,3] = PR[90,3] + 44.500;
   1:L PR[91] R[100]mm/sec CNT100;
   1:  PR[91,1] = PR[90,1] + 3.647;
   1:  PR[91,2] = PR[90,2] + 20.433;
   1:  PR[91,3] = PR[90,3] + 44.509;
   1:L PR[91] R[100]mm/sec CNT100;
   1:  PR[91,1] = PR[90,1] + 2.582;
   1:  PR[91,2] = PR[90,2] + 20.235;
   1:  PR[91,3] = PR[90,3] + 44.518;
   1:L PR[91] R[100]mm/sec CNT100;
   1:  PR[91,1] = PR[90,1] + 1.524;
   1:  PR[91,2] = PR[90,2] + 19.983;
   1:  PR[91,3] = PR[90,3] + 44.527;
   1:L PR[91] R[100]mm/sec CNT100;
   1:  PR[91,1] = PR[90,1] + 0.455;
   1:  PR[91,2] = PR[90,2] + 19.683;
   1:  PR[91,3] = PR[90,3] + 44.536;
   1:L PR[91] R[100]mm/sec CNT100;
   1:  PR[91,1] = PR[90,1] + -0.033;
   1:  PR[91,2] = PR[90,2] + 19.628;
   1:  PR[91,3] = PR[90,3] + 44.545;
   1:L PR[91] R[100]mm/sec CNT100;
   1:  PR[91,1] = PR[90,1] + -0.519;
   1:  PR[91,2] = PR[90,2] + 19.655;
   1:  PR[91,3] = PR[90,3] + 44.549;
   1:L PR[91] R[100]mm/sec CNT100;
   1:  PR[91,1] = PR[90,1] + -0.790;
   1:  PR[91,2] = PR[90,2] + 19.712;
   1:  PR[91,3] = PR[90,3] + 44.554;
   1:L PR[91] R[100]mm/sec CNT100;
   1:  PR[91,1] = PR[90,1] + -1.759;
   1:  PR[91,2] = PR[90,2] + 19.983;
   1:  PR[91,3] = PR[90,3] + 44.556;
   1:L PR[91] R[100]mm/sec CNT100;
   1:  PR[91,1] = PR[90,1] + -2.818;
   1:  PR[91,2] = PR[90,2] + 20.235;
   1:  PR[91,3] = PR[90,3] + 44.564;
   1:L PR[91] R[100]mm/sec CNT100;
   1:  PR[91,1] = PR[90,1] + -3.883;
   1:  PR[91,2] = PR[90,2] + 20.433;
   1:  PR[91,3] = PR[90,3] + 44.573;
   1:L PR[91] R[100]mm/sec CNT100;
   1:  PR[91,1] = PR[90,1] + -4.958;
   1:  PR[91,2] = PR[90,2] + 20.577;
   1:  PR[91,3] = PR[90,3] + 44.582;
   1:L PR[91] R[100]mm/sec CNT100;
   1:  PR[91,1] = PR[90,1] + -6.038;
   1:  PR[91,2] = PR[90,2] + 20.666;
   1:  PR[91,3] = PR[90,3] + 44.591;
   1:L PR[91] R[100]mm/sec CNT100;
   1:  PR[91,1] = PR[90,1] + -7.121;
   1:  PR[91,2] = PR[90,2] + 20.701;
   1:  PR[91,3] = PR[90,3] + 44.601;
   1:L PR[91] R[100]mm/sec CNT100;
   1:  PR[91,1] = PR[90,1] + -8.202;
   1:  PR[91,2] = PR[90,2] + 20.683;
   1:  PR[91,3] = PR[90,3] + 44.610;
   1:L PR[91] R[100]mm/sec CNT100;
   1:  PR[91,1] = PR[90,1] + -9.280;
   1:  PR[91,2] = PR[90,2] + 20.612;
   1:  PR[91,3] = PR[90,3] + 44.619;
   1:L PR[91] R[100]mm/sec CNT100;
   1:  PR[91,1] = PR[90,1] + -10.352;
   1:  PR[91,2] = PR[90,2] + 20.487;
   1:  PR[91,3] = PR[90,3] + 44.628;
   1:L PR[91] R[100]mm/sec CNT100;
   1:  PR[91,1] = PR[90,1] + -11.416;
   1:  PR[91,2] = PR[90,2] + 20.309;
   1:  PR[91,3] = PR[90,3] + 44.637;
   1:L PR[91] R[100]mm/sec CNT100;
   1:  PR[91,1] = PR[90,1] + -12.469;
   1:  PR[91,2] = PR[90,2] + 20.079;
   1:  PR[91,3] = PR[90,3] + 44.646;
   1:L PR[91] R[100]mm/sec CNT100;
   1:  PR[91,1] = PR[90,1] + -13.507;
   1:  PR[91,2] = PR[90,2] + 19.797;
   1:  PR[91,3] = PR[90,3] + 44.655;
   1:L PR[91] R[100]mm/sec CNT100;
   1:  PR[91,1] = PR[90,1] + -14.529;
   1:  PR[91,2] = PR[90,2] + 19.465;
   1:  PR[91,3] = PR[90,3] + 44.664;
   1:L PR[91] R[100]mm/sec CNT100;
   1:  PR[91,1] = PR[90,1] + -15.531;
   1:  PR[91,2] = PR[90,2] + 19.082;
   1:  PR[91,3] = PR[90,3] + 44.673;
   1:L PR[91] R[100]mm/sec CNT100;
   1:  PR[91,1] = PR[90,1] + -16.512;
   1:  PR[91,2] = PR[90,2] + 18.651;
   1:  PR[91,3] = PR[90,3] + 44.682;
   1:L PR[91] R[100]mm/sec CNT100;
